
// ===== library: MasterCopy "COGNEX_OUTPUTS" =====

TYPE "COGNEX_OUTPUTS"
VERSION : 0.1
   STRUCT
      Trigger_Enable : Bool;
      Trigger : Bool;
      Reserved_0 : Bool;
      Reserved_1 : Bool;
      Reserved_2 : Bool;
      Reserved_3 : Bool;
      Reserved_4 : Bool;
      Set_Offline : Bool;
      Buffer_Results_Enable : Bool;
      Inspection_Results_Ack : Bool;
      Set_User_Data : Bool;
      Reserved_5 : Bool;
      Reserved_6 : Bool;
      Reserved_7 : Bool;
      Reserved_8 : Bool;
      Reserved_9 : Bool;
      Job_Load_ID : Byte;
      Soft_Event_0 : Bool;
      Soft_Event_1 : Bool;
      Soft_Event_2 : Bool;
      Soft_Event_3 : Bool;
      Soft_Event_4 : Bool;
      Soft_Event_5 : Bool;
      Soft_Event_6 : Bool;
      Soft_Event_7 : Bool;
      User_Data : Array[1..64] of Byte;
   END_STRUCT;
END_TYPE

// ===== library: MasterCopy "COGNEX_TO_PLC" =====

TYPE "COGNEX_TO_PLC"
VERSION : 0.1
   STRUCT
      Ready : Bool;
      NOK : Bool;
      OK : Bool;
      Program_Loaded : Byte;
      Data : Array[0..63] of Byte;
   END_STRUCT;
END_TYPE

// ===== library: MasterCopy "COGNEX_INPUTS" =====

TYPE "COGNEX_INPUTS"
VERSION : 0.1
   STRUCT
      Trigger_Ready : Bool;
      Trigger_Ack : Bool;
      Acquiring : Bool;
      Missed_Acq : Bool;
      Offline_Reason_0 : Bool;
      Offline_Reason_1 : Bool;
      Offline_Reason_2 : Bool;
      Online : Bool;
      Acquisition_ID_0 : Byte;
      Acquisition_ID_1 : Byte;
      Inspecting : Bool;
      Inspection_Completed : Bool;
      Results_Buffer_Overrun : Bool;
      Results_Valid : Bool;
      Job_Loading : Bool;
      Job_Load_Complete : Bool;
      Job_Load_Failed : Bool;
      Set_User_Data_Ack : Bool;
      Job_Pass : Bool;
      Reserved_0 : Bool;
      Reserved_1 : Bool;
      Reserved_2 : Bool;
      Reserved_3 : Bool;
      Reserved_4 : Bool;
      Reserved_5 : Bool;
      Reserved_6 : Bool;
      Current_Job_ID : Byte;
      "Inspection ID_0" : Byte;
      "Inspection ID_1" : Byte;
      "Inspection Result Code" : Word;
      "Inspection Results" : Array[0..63] of Byte;
   END_STRUCT;
END_TYPE

// ===== library: MasterCopy "PLC_TO_COGNEX" =====

TYPE "PLC_TO_COGNEX"
VERSION : 0.1
   STRUCT
      Trigger : Bool;
      Change_Program : Bool;
      Program_Number : Byte;
   END_STRUCT;
END_TYPE

// ===== library: MasterCopy "Cognex_Insight_FB" =====

// folder: 3. ST1 INSPECTION/3.2. ST1 DEVICES/3.2.0. Cognex

FUNCTION_BLOCK "Cognex_Insight_FB"   // FB52, LAD
{ S7_Optimized_Access := 'FALSE' }
VERSION : 0.1
   VAR_INPUT
      Trigger : Bool;
      Change_Program : Bool;
      Program_Number : Byte;
      Inhibit : Bool;
   END_VAR
   VAR_OUTPUT
      Ready : Bool;
      OK : Bool;
      NOK : Bool;
      Program_Loaded : Byte;
      Data : Array[0..63] of Byte;
   END_VAR
   VAR
      Inspection_Completed : Bool;
      FP_Trigger : Bool;
      FP_Inspection_completed_down : Bool;
      FP_Inspection_completed_up : Bool;
      FP_Reset_Result : Bool;
      FP_Change_Program : Bool;
      NullChar : Byte;
      Outputs : "COGNEX_OUTPUTS";
      Inputs : "COGNEX_INPUTS";
   END_VAR
   VAR_TEMP
      t_DB_NO : Int;
      In_Pointer : ANY;
      Out_Pointer : ANY;
      In_Bytes_Number : Int;
      Out_Bytes_Number : Int;
      tRetVal : Int;
   END_VAR
   VAR_TEMP   // added for the SCL form of the ladder/FBD networks
      _w1 : Bool;
      _w2 : Bool;
   END_VAR
BEGIN

REGION Network 1: TRIGGER ENABLE
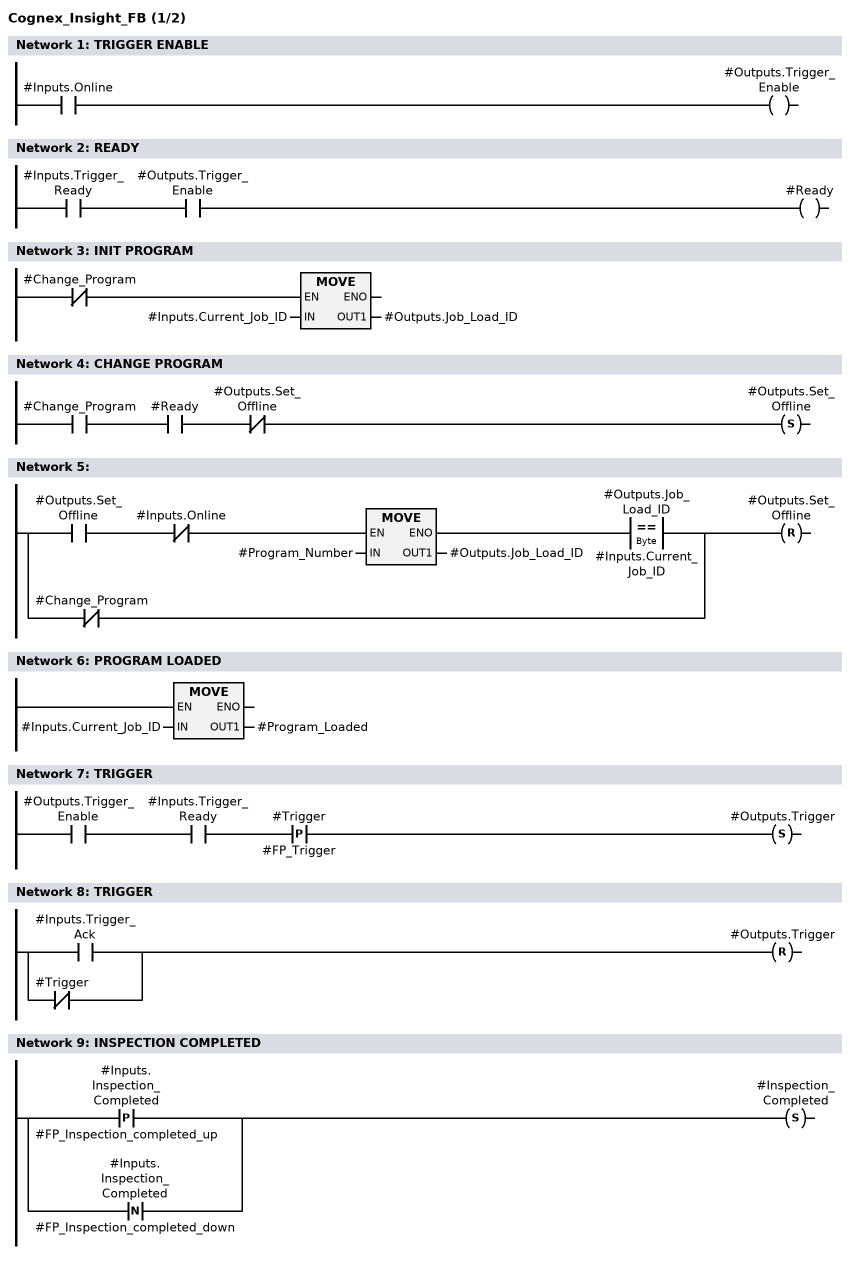
   RUNG wire#powerrail
      Contact( #Inputs.Online )
      Coil( #Outputs.Trigger_Enable )
   END_RUNG
   // the same network as SCL:
   #Outputs.Trigger_Enable := #Inputs.Online;
END_REGION

REGION Network 2: READY
   RUNG wire#powerrail
      Contact( #Inputs.Trigger_Ready )
      Contact( #Outputs.Trigger_Enable )
      Coil( #Ready )
   END_RUNG
   // the same network as SCL:
   #Ready := #Inputs.Trigger_Ready AND #Outputs.Trigger_Enable;
END_REGION

REGION Network 3: INIT PROGRAM
   RUNG wire#powerrail
      I_Contact( #Change_Program )
      { S7_GenerateENO := "TRUE" } Move(in := #Inputs.Current_Job_ID, out1 => #Outputs.Job_Load_ID)
   END_RUNG
   // the same network as SCL:
   IF NOT #Change_Program THEN #Outputs.Job_Load_ID := #Inputs.Current_Job_ID; END_IF;
END_REGION

REGION Network 4: CHANGE PROGRAM
   RUNG wire#powerrail
      Contact( #Change_Program )
      Contact( #Ready )
      I_Contact( #Outputs.Set_Offline )
      S_Coil( #Outputs.Set_Offline )
   END_RUNG
   // the same network as SCL:
   IF #Change_Program AND #Ready AND NOT #Outputs.Set_Offline THEN #Outputs.Set_Offline := TRUE; END_IF;
END_REGION

REGION Network 5
   RUNG wire#powerrail
      Contact( #Outputs.Set_Offline )
      I_Contact( #Inputs.Online )
      { S7_GenerateENO := "TRUE" } Move(in := #Program_Number, out1 => #Outputs.Job_Load_ID)
      { S7_Templates := "SrcType := Byte" } EQ_Contact(in1 := #Outputs.Job_Load_ID, in2 := #Inputs.Current_Job_ID)
      wire#w1
      R_Coil( #Outputs.Set_Offline )
   END_RUNG
   RUNG wire#powerrail
      I_Contact( #Change_Program )
   END_RUNG wire#w1
   // the same network as SCL:
   // ENO of a box is taken as its EN; it also drops when the box reports an error
   #_w1 := #Outputs.Set_Offline AND NOT #Inputs.Online;
   IF #_w1 THEN #Outputs.Job_Load_ID := #Program_Number; END_IF;
   IF (#_w1 AND (#Outputs.Job_Load_ID = #Inputs.Current_Job_ID)) OR NOT #Change_Program THEN
       #Outputs.Set_Offline := FALSE;
   END_IF;
END_REGION

REGION Network 6: PROGRAM LOADED
   RUNG wire#powerrail
      { S7_GenerateENO := "TRUE" } Move(in := #Inputs.Current_Job_ID, out1 => #Program_Loaded)
   END_RUNG
   // the same network as SCL:
   #Program_Loaded := #Inputs.Current_Job_ID;
END_REGION

REGION Network 7: TRIGGER
   RUNG wire#powerrail
      Contact( #Outputs.Trigger_Enable )
      Contact( #Inputs.Trigger_Ready )
      P_Contact(operand := #Trigger, bit := #FP_Trigger)
      S_Coil( #Outputs.Trigger )
   END_RUNG
   // the same network as SCL:
   #_w1 := #Outputs.Trigger_Enable AND #Inputs.Trigger_Ready AND #Trigger AND NOT #FP_Trigger;   // rising edge of #Trigger
   #FP_Trigger := #Trigger;
   IF #_w1 THEN #Outputs.Trigger := TRUE; END_IF;
END_REGION

REGION Network 8: TRIGGER
   RUNG wire#powerrail
      Contact( #Inputs.Trigger_Ack )
      wire#w1
      R_Coil( #Outputs.Trigger )
   END_RUNG
   RUNG wire#powerrail
      I_Contact( #Trigger )
   END_RUNG wire#w1
   // the same network as SCL:
   IF #Inputs.Trigger_Ack OR NOT #Trigger THEN #Outputs.Trigger := FALSE; END_IF;
END_REGION

REGION Network 9: INSPECTION COMPLETED
   RUNG wire#powerrail
      P_Contact(operand := #Inputs.Inspection_Completed, bit := #FP_Inspection_completed_up)
      wire#w1
      S_Coil( #Inspection_Completed )
   END_RUNG
   RUNG wire#powerrail
      N_Contact(operand := #Inputs.Inspection_Completed, bit := #FP_Inspection_completed_down)
   END_RUNG wire#w1
   // the same network as SCL:
   #_w1 := #Inputs.Inspection_Completed AND NOT #FP_Inspection_completed_up;   // rising edge of #Inputs.Inspection_Completed
   #FP_Inspection_completed_up := #Inputs.Inspection_Completed;
   #_w2 := NOT #Inputs.Inspection_Completed AND #FP_Inspection_completed_down;   // falling edge of #Inputs.Inspection_Completed
   #FP_Inspection_completed_down := #Inputs.Inspection_Completed;
   IF #_w1 OR #_w2 THEN #Inspection_Completed := TRUE; END_IF;
END_REGION

REGION Network 10: OK/NOK AND DATA / OK/NOK
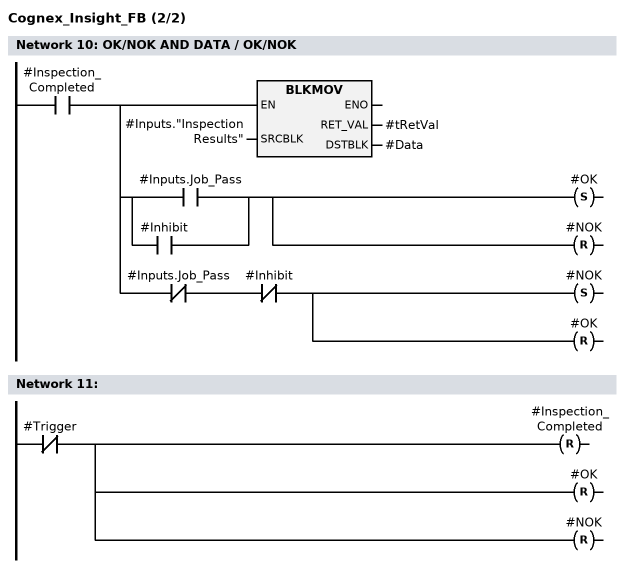
   IF #Inspection_Completed THEN
       #tRetVal := BLKMOV(SRCBLK := #Inputs."Inspection Results", DSTBLK => #Data);
   END_IF;
   IF #Inspection_Completed AND (#Inputs.Job_Pass OR #Inhibit) THEN
       #OK := TRUE;
       #NOK := FALSE;
   END_IF;
   IF #Inspection_Completed AND NOT #Inputs.Job_Pass AND NOT #Inhibit THEN
       #NOK := TRUE;
       #OK := FALSE;
   END_IF;
END_REGION

REGION Network 11
   RUNG wire#powerrail
      I_Contact( #Trigger )
      wire#w1
      R_Coil( #Inspection_Completed )
   END_RUNG
   RUNG wire#w1
      R_Coil( #OK )
   END_RUNG
   RUNG wire#w1
      R_Coil( #NOK )
   END_RUNG
   // the same network as SCL:
   IF NOT #Trigger THEN
       #Inspection_Completed := FALSE;
       #OK := FALSE;
       #NOK := FALSE;
   END_IF;
END_REGION

REGION Network 12: FUNCTION OUT
END_REGION
END_FUNCTION_BLOCK

// ===== library: MasterCopy "Keyence_SR1000_FB" =====

// folder: 3. ST1 INSPECTION/3.2. ST1 DEVICES/3.2.1. Keyence

FUNCTION_BLOCK "Keyence_SR1000_FB"   // FB59, LAD
{ S7_Optimized_Access := 'FALSE' }
VERSION : 0.1
   VAR_INPUT
      Trigger : Bool;
      Clear_Error : Bool;
      Inhibit : Bool;
   END_VAR
   VAR_OUTPUT
      Ready : Bool;
      Error : Bool;
      Error_Code : Word;
      Ok : Bool;
      NOK : Bool;
      Data : Array[0..26] of Byte;
   END_VAR
   VAR
      Inputs : "SR1000_IN";
      Outputs : "SR1000_OUT";
      "Blank Data" : Array[0..26] of Byte;
      Trigger_Flank : Bool;
      t_timeout : TON;
      s_timeout_error : Bool;
   END_VAR
   VAR_TEMP
      retval : Int;
   END_VAR
   VAR_TEMP   // added for the SCL form of the ladder/FBD networks
      _w1 : Bool;
      _w2 : Bool;
   END_VAR
BEGIN

REGION Network 1: ////////INPUTS//////////////////////
END_REGION

REGION Network 2: Ready
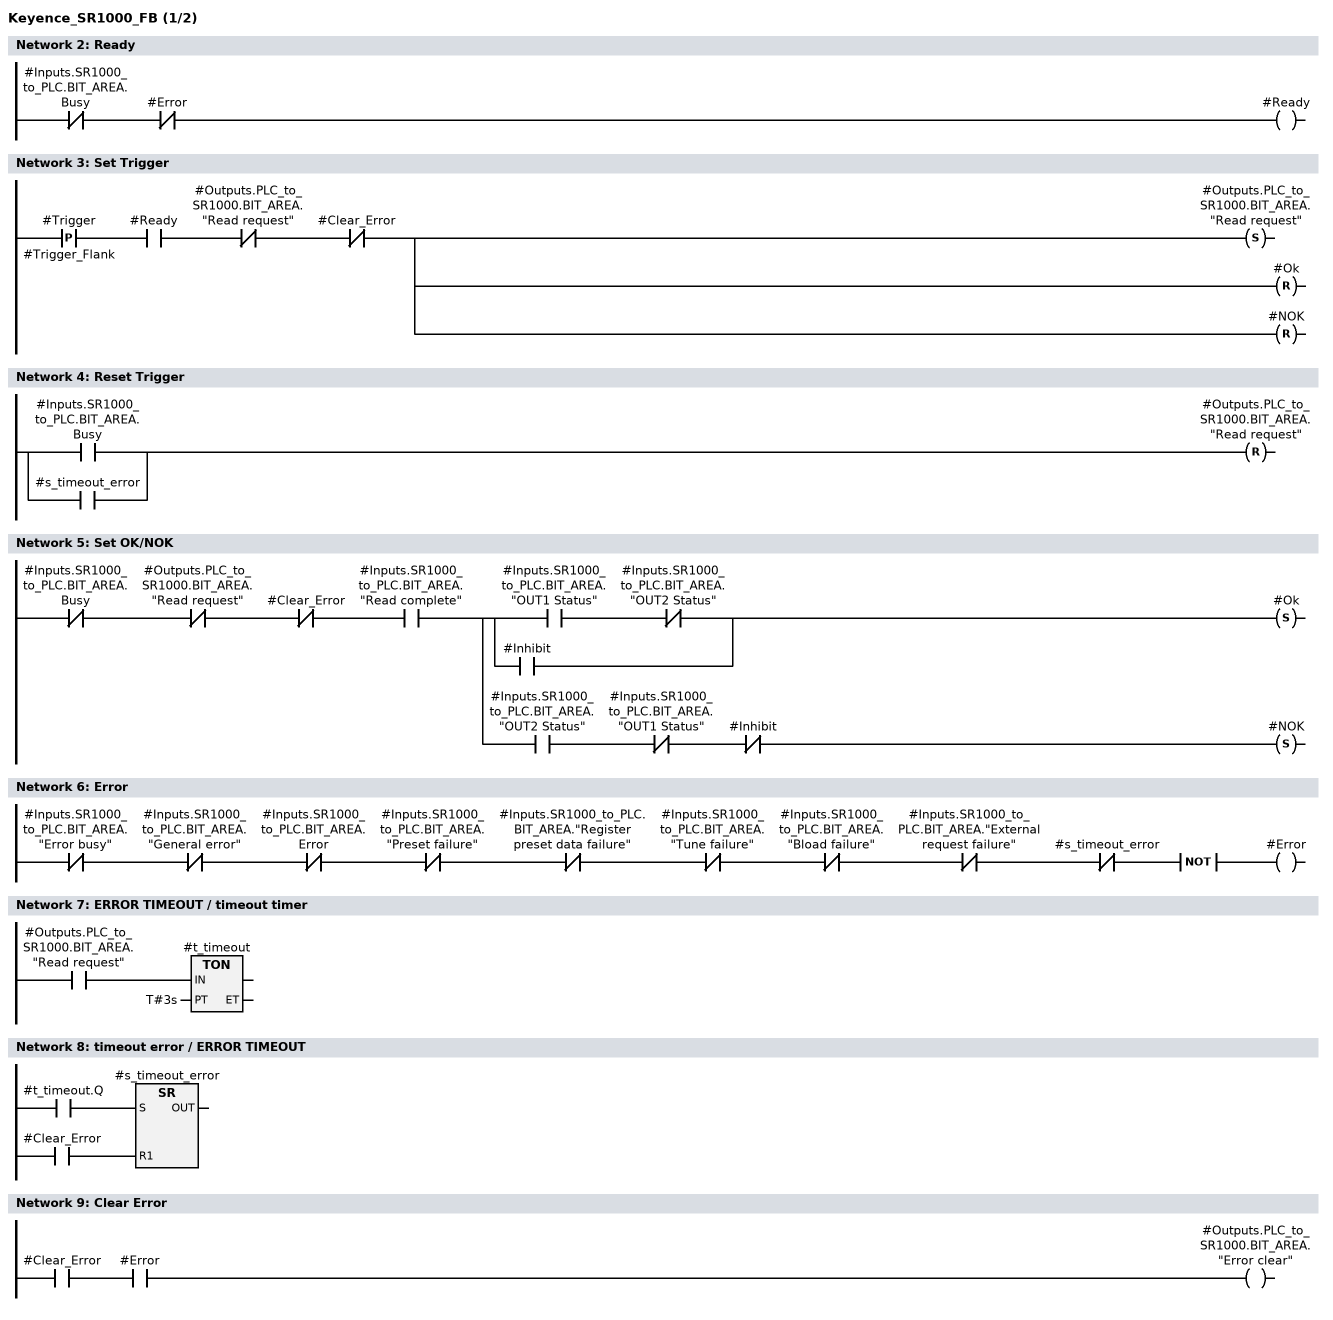
   RUNG wire#powerrail
      I_Contact( #Inputs.SR1000_to_PLC.BIT_AREA.Busy )
      I_Contact( #Error )
      Coil( #Ready )
   END_RUNG
   // the same network as SCL:
   #Ready := NOT #Inputs.SR1000_to_PLC.BIT_AREA.Busy AND NOT #Error;
END_REGION

REGION Network 3: Set Trigger
   RUNG wire#powerrail
      P_Contact(operand := #Trigger, bit := #Trigger_Flank)
      Contact( #Ready )
      I_Contact( #Outputs.PLC_to_SR1000.BIT_AREA."Read request" )
      I_Contact( #Clear_Error )
      wire#w1
      S_Coil( #Outputs.PLC_to_SR1000.BIT_AREA."Read request" )
   END_RUNG
   RUNG wire#w1
      R_Coil( #Ok )
   END_RUNG
   RUNG wire#w1
      R_Coil( #NOK )
   END_RUNG
   // the same network as SCL:
   #_w1 := #Trigger AND NOT #Trigger_Flank;   // rising edge of #Trigger
   #Trigger_Flank := #Trigger;
   #_w2 := #_w1 AND #Ready AND NOT #Outputs.PLC_to_SR1000.BIT_AREA."Read request" AND NOT #Clear_Error;
   IF #_w2 THEN
       #Outputs.PLC_to_SR1000.BIT_AREA."Read request" := TRUE;
       #Ok := FALSE;
       #NOK := FALSE;
   END_IF;
END_REGION

REGION Network 4: Reset Trigger
   RUNG wire#powerrail
      Contact( #Inputs.SR1000_to_PLC.BIT_AREA.Busy )
      wire#w1
      R_Coil( #Outputs.PLC_to_SR1000.BIT_AREA."Read request" )
   END_RUNG
   RUNG wire#powerrail
      Contact( #s_timeout_error )
   END_RUNG wire#w1
   // the same network as SCL:
   IF #Inputs.SR1000_to_PLC.BIT_AREA.Busy OR #s_timeout_error THEN
       #Outputs.PLC_to_SR1000.BIT_AREA."Read request" := FALSE;
   END_IF;
END_REGION

REGION Network 5: Set OK/NOK
   RUNG wire#powerrail
      I_Contact( #Inputs.SR1000_to_PLC.BIT_AREA.Busy )
      I_Contact( #Outputs.PLC_to_SR1000.BIT_AREA."Read request" )
      I_Contact( #Clear_Error )
      Contact( #Inputs.SR1000_to_PLC.BIT_AREA."Read complete" )
      wire#w1
      Contact( #Inputs.SR1000_to_PLC.BIT_AREA."OUT1 Status" )
      I_Contact( #Inputs.SR1000_to_PLC.BIT_AREA."OUT2 Status" )
      wire#w2
      S_Coil( #Ok )
   END_RUNG
   RUNG wire#w1
      Contact( #Inhibit )
   END_RUNG wire#w2
   RUNG wire#w1
      Contact( #Inputs.SR1000_to_PLC.BIT_AREA."OUT2 Status" )
      I_Contact( #Inputs.SR1000_to_PLC.BIT_AREA."OUT1 Status" )
      I_Contact( #Inhibit )
      S_Coil( #NOK )
   END_RUNG
   // the same network as SCL:
   #_w1 := NOT #Inputs.SR1000_to_PLC.BIT_AREA.Busy AND NOT #Outputs.PLC_to_SR1000.BIT_AREA."Read request" AND NOT #Clear_Error AND #Inputs.SR1000_to_PLC.BIT_AREA."Read complete";
   IF #_w1 AND ((#Inputs.SR1000_to_PLC.BIT_AREA."OUT1 Status" AND NOT #Inputs.SR1000_to_PLC.BIT_AREA."OUT2 Status") OR #Inhibit) THEN
       #Ok := TRUE;
   END_IF;
   IF #_w1 AND #Inputs.SR1000_to_PLC.BIT_AREA."OUT2 Status" AND NOT #Inputs.SR1000_to_PLC.BIT_AREA."OUT1 Status" AND NOT #Inhibit THEN
       #NOK := TRUE;
   END_IF;
END_REGION

REGION Network 6: Error
   RUNG wire#powerrail
      I_Contact( #Inputs.SR1000_to_PLC.BIT_AREA."Error busy" )
      I_Contact( #Inputs.SR1000_to_PLC.BIT_AREA."General error" )
      I_Contact( #Inputs.SR1000_to_PLC.BIT_AREA.Error )
      I_Contact( #Inputs.SR1000_to_PLC.BIT_AREA."Preset failure" )
      I_Contact( #Inputs.SR1000_to_PLC.BIT_AREA."Register preset data failure" )
      I_Contact( #Inputs.SR1000_to_PLC.BIT_AREA."Tune failure" )
      I_Contact( #Inputs.SR1000_to_PLC.BIT_AREA."Bload failure" )
      I_Contact( #Inputs.SR1000_to_PLC.BIT_AREA."External request failure" )
      I_Contact( #s_timeout_error )
      Not()
      Coil( #Error )
   END_RUNG
   // the same network as SCL:
   #Error := NOT (NOT #Inputs.SR1000_to_PLC.BIT_AREA."Error busy" AND NOT #Inputs.SR1000_to_PLC.BIT_AREA."General error" AND NOT #Inputs.SR1000_to_PLC.BIT_AREA.Error AND NOT #Inputs.SR1000_to_PLC.BIT_AREA."Preset failure" AND NOT #Inputs.SR1000_to_PLC.BIT_AREA."Register preset data failure" AND NOT #Inputs.SR1000_to_PLC.BIT_AREA."Tune failure" AND NOT #Inputs.SR1000_to_PLC.BIT_AREA."Bload failure" AND NOT #Inputs.SR1000_to_PLC.BIT_AREA."External request failure" AND NOT #s_timeout_error);
END_REGION

REGION Network 7: ERROR TIMEOUT / timeout timer
   #t_timeout.TON(IN := #Outputs.PLC_to_SR1000.BIT_AREA."Read request", PT := T#3s);
END_REGION

REGION Network 8: timeout error / ERROR TIMEOUT
   RUNG wire#powerrail
      Contact( #t_timeout.Q )
      S_SR(operand := #s_timeout_error, r1 := wire#w1)
   END_RUNG
   RUNG wire#powerrail
      Contact( #Clear_Error )
   END_RUNG wire#w1
   // the same network as SCL:
   IF #t_timeout.Q THEN
       #s_timeout_error := TRUE;   // SR flip-flop
   END_IF;
   IF #Clear_Error THEN #s_timeout_error := FALSE; END_IF;
END_REGION

REGION Network 9: Clear Error
   RUNG wire#powerrail
      Contact( #Clear_Error )
      Contact( #Error )
      Coil( #Outputs.PLC_to_SR1000.BIT_AREA."Error clear" )
   END_RUNG
   // the same network as SCL:
   #Outputs.PLC_to_SR1000.BIT_AREA."Error clear" := #Clear_Error AND #Error;
END_REGION

REGION Network 10: Transfer Data
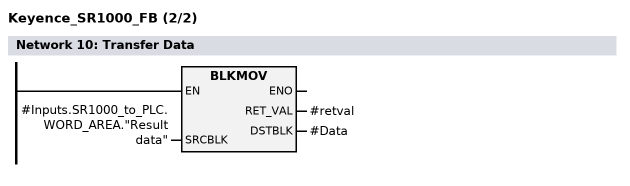
   #retval := BLKMOV(SRCBLK := #Inputs.SR1000_to_PLC.WORD_AREA."Result data", DSTBLK => #Data);
END_REGION
END_FUNCTION_BLOCK

// ===== library: MasterCopy "KEYENCE_TO_PLC" =====

TYPE "KEYENCE_TO_PLC"
   STRUCT
      Ready : Bool;
      Error : Bool;
      ErrorCode : Word;
      OK : Bool;
      NOK : Bool;
      Data : Array[0..26] of Byte;
   END_STRUCT;
END_TYPE

// ===== library: MasterCopy "PLC_TO_KEYENCE" =====

TYPE "PLC_TO_KEYENCE"
   STRUCT
      Trigger : Bool;
      "Clear Data" : Bool;
      "Clear Error" : Bool;
   END_STRUCT;
END_TYPE

// ===== library: MasterCopy "SR1000_IN" =====

TYPE "SR1000_IN"
VERSION : 0.1
   STRUCT
      SR1000_to_PLC : Struct
         BIT_AREA : Struct
            Error : Bool;   // Error
            "Result data available" : Bool;   // Result data available
            "Result data strobe" : Bool := false;   // Result data strobe
            DBX_0_3 : Bool := false;
            DBX_0_4 : Bool := false;
            DBX_0_5 : Bool := false;
            "Buffer overflow error" : Bool := false;   // Buffer overflow error
            "General error" : Bool := false;   // General error
            Busy : Bool := false;   // Busy
            "Trg busy" : Bool := false;   // Trg busy
            "Lock busy" : Bool := false;   // Lock busy
            "Mode busy" : Bool := false;   // Mode busy
            "Error busy" : Bool := false;   // Error busy
            DBX_1_5 : Bool := false;
            DBX_1_6 : Bool := false;
            DBX_1_7 : Bool := false;
            "Read complete" : Bool := false;   // Read complete
            "Preset complete" : Bool := false;   // Preset complete
            "Register preset data complete" : Bool := false;   // Register preset data complete
            "Tune complete" : Bool := false;   // Tune complete
            "Bload complete" : Bool := false;   // Bload complete
            DBX_2_5 : Bool := false;
            DBX_2_6 : Bool := false;
            "External request complete" : Bool := false;   // External request complete
            "Read failure" : Bool := false;   // Read failure
            "Preset failure" : Bool := false;   // Preset failure
            "Register preset data failure" : Bool := false;   // Register preset data failure
            "Tune failure" : Bool := false;   // Tune failure
            "Bload failure" : Bool := false;   // Bload failure
            DBX_3_5 : Bool := false;
            DBX_3_6 : Bool := false;
            "External request failure" : Bool := false;   // External request failure
            "IN1 Status" : Bool := false;   // IN1 Status
            "IN2 Status" : Bool := false;   // IN2 Status
            DBX_4_2 : Bool := false;
            DBX_4_3 : Bool := false;
            "OUT1 Status" : Bool := false;   // OUT1 Status
            "OUT2 Status" : Bool := false;   // OUT2 Status
            "OUT3 Status" : Bool := false;   // OUT3 Status
            DBX_4_7 : Bool := false;
            Unstable : Bool := false;   // Unstable
            "Matching level unstable" : Bool := false;   // Matching level unstable
            "ISO/IEC15415 unstable" : Bool := false;   // ISO/IEC15415 unstable
            "AIM DPM unstable" : Bool := false;   // AIM DPM unstable
            "SAE AS9132 unstable" : Bool := false;   // SAE AS9132 unstable
            DBX_5_5 : Bool := false;
            DBX_5_6 : Bool := false;
            DBX_5_7 : Bool := false;
         END_STRUCT;
         WORD_AREA : Struct
            "Matching level" : Word;   // Matching level
            "ISO/IEC 15415 grade" : Word;   // ISO/IEC 15415 grade
            "AIM DPM Grade" : Word;   // AIM DPM Grade
            DBW_7_3 : Word;
            "Read result code" : Word;   // Read result code
            "Preset result code" : Word;   // Preset result code
            "Register preset data result code" : Word;   // Register preset data result code
            "Tune result code" : Word;   // Tune result code
            "Bload result code" : Word;   // Bload result code
            DBW_8_5 : Word;
            DBW_8_6 : Word;
            "Ext. request result code" : Word;   // Ext. request result code
            "General error code" : Word;   // General error code
            "Slave ID" : Word;   // Slave ID
            "Result data ready count" : Word;   // Result data ready count
            "Result data update count" : Word;   // Result data update count
            "Trigger input count for master" : Word;   // Trigger input count for master
            DBW_9_4 : Byte;   // Result data size
            "Result data size" : Byte;
            "Result data" : Array[1..128] of Byte;   // Result data
         END_STRUCT;
      END_STRUCT;
   END_STRUCT;
END_TYPE

// ===== library: MasterCopy "SR1000_OUT" =====

TYPE "SR1000_OUT"
VERSION : 0.1
   STRUCT
      PLC_to_SR1000 : Struct
         BIT_AREA : Struct
            DBX170_0 : Bool;
            "Result data latch" : Bool := false;   // Result data latch
            DBX170_2 : Bool := false;
            DBX170_3 : Bool := false;
            DBX170_4 : Bool := false;
            DBX170_5 : Bool := false;
            DBX170_6 : Bool := false;
            "Error clear" : Bool := false;   // Error clear
            "Read request" : Bool := false;   // Read request
            "Preset request" : Bool := false;   // Preset request
            "Register preset" : Bool := false;   // Register preset
            "Tune request" : Bool := false;   // Tune request
            "Bload request" : Bool := false;   // Bload request
            DBX171_5 : Bool := false;
            DBX171_6 : Bool := false;
            DBX171_7 : Bool := false;
            "Read complete clear" : Bool := false;   // Read complete clear
            "Preset complet clear" : Bool := false;   // Preset complet clear
            "Register preset data complete clear" : Bool := false;   // Register preset data complete clear
            "Tune complete clear" : Bool := false;   // Tune complete clear
            "Bload complete clear" : Bool := false;   // Bload complete clear
            DBX172_5 : Bool := false;
            DBX172_6 : Bool := false;
            "External request complete clear" : Bool := false;   // External request complete clear
            "Bank number\Bload file number" : Word;   // Bank number\Bload file number
            "User data size" : Word := 16#0;   // User data size
            "User data" : Array[1..128] of Byte;   // User data
         END_STRUCT;
      END_STRUCT;
   END_STRUCT;
END_TYPE

// ===== library: MasterCopy "DATAMAN_TO_PLC" =====

TYPE "DATAMAN_TO_PLC"
VERSION : 0.1
   STRUCT
      Ready : Bool;
      Trigger_ACK : Bool;
      OK : Bool;
      NOK : Bool;
      Error : Bool;
      Result_ID : Word;
      Result_Lenght : Int;
      Result : Array[1..64] of Byte;
   END_STRUCT;
END_TYPE

// ===== library: MasterCopy "DATAMAN_INPUTS" =====

TYPE "DATAMAN_INPUTS"
VERSION : 0.1
   STRUCT
      Trigger_Ready : Bool;
      Trigger_Ack : Bool;
      Acquiring : Bool;
      Missed_Acq : Bool;
      Reserved_0 : Bool;
      Reserved_1 : Bool;
      Reserved_2 : Bool;
      Reserved_3 : Bool;
      Trigger_ID_0 : Byte;
      Trigger_ID_1 : Byte;
      Decoding : Bool;
      Decode_Complete : Bool;
      Result_Buffer_Overrun : Bool;
      Result_Available : Bool;
      Reserved_4 : Bool;
      Reserved_5 : Bool;
      Reserved_6 : Bool;
      General_Fault : Bool;
      Train_Code_Ack : Bool;
      Train_Match_String_Ack : Bool;
      Train_Focus_Ack : Bool;
      Train_Brightness_Ack : Bool;
      Ultrain_Ack : Bool;
      Reserved_7 : Bool;
      Execute_DMCC_Ack : Bool;
      Set_Match_String_Ack : Bool;
      Result_ID_0 : Byte;
      Result_ID_1 : Byte;
      Result_Code_0 : Byte;
      Result_Code_1 : Byte;
      Result_Extended_0 : Byte;
      Result_Extended_1 : Byte;
      Result_Length_0 : Byte;
      Result_Length_1 : Byte;
      Result_Data_0 : Byte;
      Result_Data_1 : Byte;
      Result_Data_2 : Byte;
      Result_Data_3 : Byte;
      Result_Data_4 : Byte;
      Result_Data_5 : Byte;
      Result_Data_6 : Byte;
      Result_Data_7 : Byte;
      Result_Data_8 : Byte;
      Result_Data_9 : Byte;
      Result_Data_10 : Byte;
      Result_Data_11 : Byte;
      Result_Data_12 : Byte;
      Result_Data_13 : Byte;
      Result_Data_14 : Byte;
      Result_Data_15 : Byte;
      Result_Data_16 : Byte;
      Result_Data_17 : Byte;
      Result_Data_18 : Byte;
      Result_Data_19 : Byte;
      Result_Data_20 : Byte;
      Result_Data_21 : Byte;
      Result_Data_22 : Byte;
      Result_Data_23 : Byte;
      Result_Data_24 : Byte;
      Result_Data_25 : Byte;
      Result_Data_26 : Byte;
      Result_Data_27 : Byte;
      Result_Data_28 : Byte;
      Result_Data_29 : Byte;
      Result_Data_30 : Byte;
      Result_Data_31 : Byte;
      Result_Data_32 : Byte;
      Result_Data_33 : Byte;
      Result_Data_34 : Byte;
      Result_Data_35 : Byte;
      Result_Data_36 : Byte;
      Result_Data_37 : Byte;
      Result_Data_38 : Byte;
      Result_Data_39 : Byte;
      Result_Data_40 : Byte;
      Result_Data_41 : Byte;
      Result_Data_42 : Byte;
      Result_Data_43 : Byte;
      Result_Data_44 : Byte;
      Result_Data_45 : Byte;
      Result_Data_46 : Byte;
      Result_Data_47 : Byte;
      Result_Data_48 : Byte;
      Result_Data_49 : Byte;
      Result_Data_50 : Byte;
      Result_Data_51 : Byte;
      Result_Data_52 : Byte;
      Result_Data_53 : Byte;
      Result_Data_54 : Byte;
      Result_Data_55 : Byte;
      Result_Data_56 : Byte;
      Result_Data_57 : Byte;
      Result_Data_58 : Byte;
      Result_Data_59 : Byte;
      Result_Data_60 : Byte;
      Result_Data_61 : Byte;
      Result_Data_62 : Byte;
      Result_Data_63 : Byte;
   END_STRUCT;
END_TYPE

// ===== library: MasterCopy "DATAMAN_OUTPUTS" =====

TYPE "DATAMAN_OUTPUTS"
VERSION : 0.1
   STRUCT
      Trigger_Enable : Bool;
      Trigger : Bool;
      Reserved_0 : Bool;
      Reserved_1 : Bool;
      Reserved_2 : Bool;
      Reserved_3 : Bool;
      Reserved_4 : Bool;
      Reserved_5 : Bool;
      Result_Buffer_Enable : Bool;
      Results_Ack : Bool;
      Reserved_6 : Bool;
      Reserved_7 : Bool;
      Reserved_8 : Bool;
      Reserved_9 : Bool;
      Reserved_10 : Bool;
      Reserved_11 : Bool;
      Train_Code : Bool;
      Train_Match_String : Bool;
      Train_Focus : Bool;
      Train_Brightness : Bool;
      Ultrain : Bool;
      Reserved_12 : Bool;
      Execute_DMCC : Bool;
      Set_Match_String : Bool;
      User_Data_Option_0 : Byte;
      User_Data_Option_1 : Byte;
      User_Data_Lenght_0 : Byte;
      User_Data_Lenght_1 : Byte;
      User_Data_0 : Byte;
      User_Data_1 : Byte;
      User_Data_2 : Byte;
      User_Data_3 : Byte;
      User_Data_4 : Byte;
      User_Data_5 : Byte;
      User_Data_6 : Byte;
      User_Data_7 : Byte;
      User_Data_8 : Byte;
      User_Data_9 : Byte;
      User_Data_10 : Byte;
      User_Data_11 : Byte;
      User_Data_12 : Byte;
      User_Data_13 : Byte;
      User_Data_14 : Byte;
      User_Data_15 : Byte;
      User_Data_16 : Byte;
      User_Data_17 : Byte;
      User_Data_18 : Byte;
      User_Data_19 : Byte;
      User_Data_20 : Byte;
      User_Data_21 : Byte;
      User_Data_22 : Byte;
      User_Data_23 : Byte;
      User_Data_24 : Byte;
      User_Data_25 : Byte;
      User_Data_26 : Byte;
      User_Data_27 : Byte;
      User_Data_28 : Byte;
      User_Data_29 : Byte;
      User_Data_30 : Byte;
      User_Data_31 : Byte;
      User_Data_32 : Byte;
      User_Data_33 : Byte;
      User_Data_34 : Byte;
      User_Data_35 : Byte;
      User_Data_36 : Byte;
      User_Data_37 : Byte;
      User_Data_38 : Byte;
      User_Data_39 : Byte;
      User_Data_40 : Byte;
      User_Data_41 : Byte;
      User_Data_42 : Byte;
      User_Data_43 : Byte;
      User_Data_44 : Byte;
      User_Data_45 : Byte;
      User_Data_46 : Byte;
      User_Data_47 : Byte;
      User_Data_48 : Byte;
      User_Data_49 : Byte;
      User_Data_50 : Byte;
      User_Data_51 : Byte;
      User_Data_52 : Byte;
      User_Data_53 : Byte;
      User_Data_54 : Byte;
      User_Data_55 : Byte;
      User_Data_56 : Byte;
      User_Data_57 : Byte;
      User_Data_58 : Byte;
      User_Data_59 : Byte;
      User_Data_60 : Byte;
      User_Data_61 : Byte;
      User_Data_62 : Byte;
      User_Data_63 : Byte;
   END_STRUCT;
END_TYPE

// ===== library: MasterCopy "PLC_TO_DATAMAN" =====

TYPE "PLC_TO_DATAMAN"
VERSION : 0.1
   STRUCT
      Reset : Bool;
      Result_Ack : Bool;
   END_STRUCT;
END_TYPE

// ===== library: MasterCopy "Dataman_FB" =====

// folder: 8. DRAWERS/8.2. ST6 DEVICES/8.2.1.Dataman

FUNCTION_BLOCK "Dataman_FB"   // FB51, LAD
{ S7_Optimized_Access := 'FALSE' }
VERSION : 0.1
   VAR_INPUT
      Reset : Bool;
      I_O_Address : Int;   // dirección entradas salidas en configuración de hardware
      DB_NO : Int;   // Número del db de instancia
   END_VAR
   VAR_OUTPUT
      Ready : Bool;
      Trigger_ACK : Bool;
      OK : Bool;
      NOK : Bool;
      Error : Bool;
      Result_ID : Word;
      Result_Lenght : Int;
      Result : Array[1..64] of Byte;
   END_VAR
   VAR
      WaitingNewTrigger : Bool;
      ResultAckPending : Bool;
      Result_Code : Word;
      Inputs : "DATAMAN_INPUTS";
      Outputs : "DATAMAN_OUTPUTS";
   END_VAR
   VAR_TEMP
      On : Bool;
      Off : Bool;
      t_DB_NO : Int;
      In_Pointer : ANY;
      Outputs_Bytes_Number : Int;
      Inputs_Bytes_Number : Int;
      Out_Pointer : ANY;
      tRetVal : Int;
   END_VAR
   VAR_TEMP   // added for the SCL form of the ladder/FBD networks
      _w1 : Bool;
   END_VAR
BEGIN

REGION Network 1
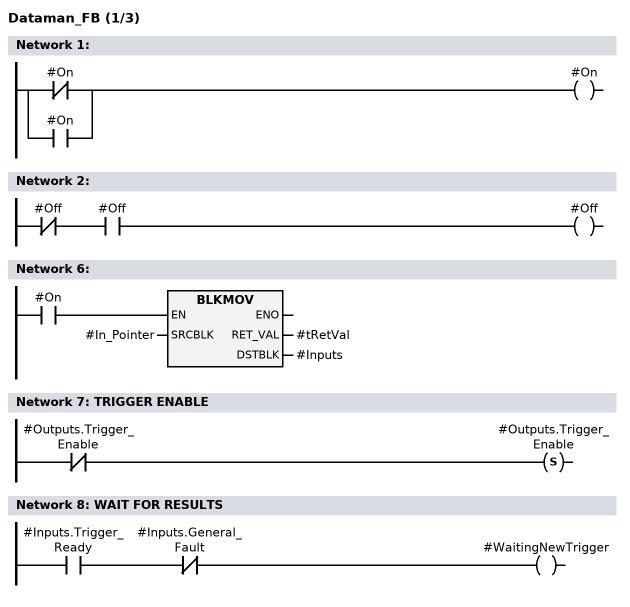
   RUNG wire#powerrail
      I_Contact( #On )
      wire#w1
      Coil( #On )
   END_RUNG
   RUNG wire#powerrail
      Contact( #On )
   END_RUNG wire#w1
   // the same network as SCL:
   #On := NOT #On OR #On;
END_REGION

REGION Network 2
   RUNG wire#powerrail
      I_Contact( #Off )
      Contact( #Off )
      Coil( #Off )
   END_RUNG
   // the same network as SCL:
   #Off := NOT #Off AND #Off;
END_REGION

REGION Network 3 (STL)

         L     #DB_NO;
         T     #t_DB_NO;
         OPN   DB[ #t_DB_NO];
END_REGION

REGION Network 4 (STL)

         L     77;
         T     #Inputs_Bytes_Number;
END_REGION

REGION Network 5 (STL)
   //En primer lugar, apuntar al puntero
         LAR1;
   //Carga de parámetros en los bytes del puntero
   //Byte 0 = 10h para S7
         L     16#10;
         T     LB[AR1, P#0.0];

   //Byte 1 = Tipo de datos
   //02h para byte
         L     16#02;
         T     LB[AR1, P#1.0];

   //Byte2-Byte3 (int) = Factor de repetición
   //número de bytes (tipo de datos) a mover
         L     #Inputs_Bytes_Number;
         T     LW[AR1, P#2.0];

   //Byt42-Byte5 (int) = Número de DB
   //0 en este caso porque no se trata de DB
         L     0;
         T     LW[AR1, P#4.0];

   //En los siguientes 4 bytes van el area de memoria y la dirección inicial
   //Se borra inicialmente
         L     0;
         T     LD[AR1, P#6.0];

   //Byte 6 = Area de memoria
   //81h para entradas
         L     16#81;
         T     LB[AR1, P#6.0];


   //Byte7-Byte9 (int) = dirección (byte.bit)
   //ver formato
         L     #I_O_Address;
         SLW   3;
         T     LW[AR1, P#8.0];
END_REGION

REGION Network 6
   IF #On THEN #tRetVal := BLKMOV(SRCBLK := #In_Pointer, DSTBLK => #Inputs); END_IF;
END_REGION

REGION Network 7: TRIGGER ENABLE
   RUNG wire#powerrail
      I_Contact( #Outputs.Trigger_Enable )
      S_Coil( #Outputs.Trigger_Enable )
   END_RUNG
   // the same network as SCL:
   IF NOT #Outputs.Trigger_Enable THEN #Outputs.Trigger_Enable := TRUE; END_IF;
END_REGION

REGION Network 8: WAIT FOR RESULTS
   RUNG wire#powerrail
      Contact( #Inputs.Trigger_Ready )
      I_Contact( #Inputs.General_Fault )
      Coil( #WaitingNewTrigger )
   END_RUNG
   // the same network as SCL:
   #WaitingNewTrigger := #Inputs.Trigger_Ready AND NOT #Inputs.General_Fault;
END_REGION

REGION Network 9: SAVE DATA
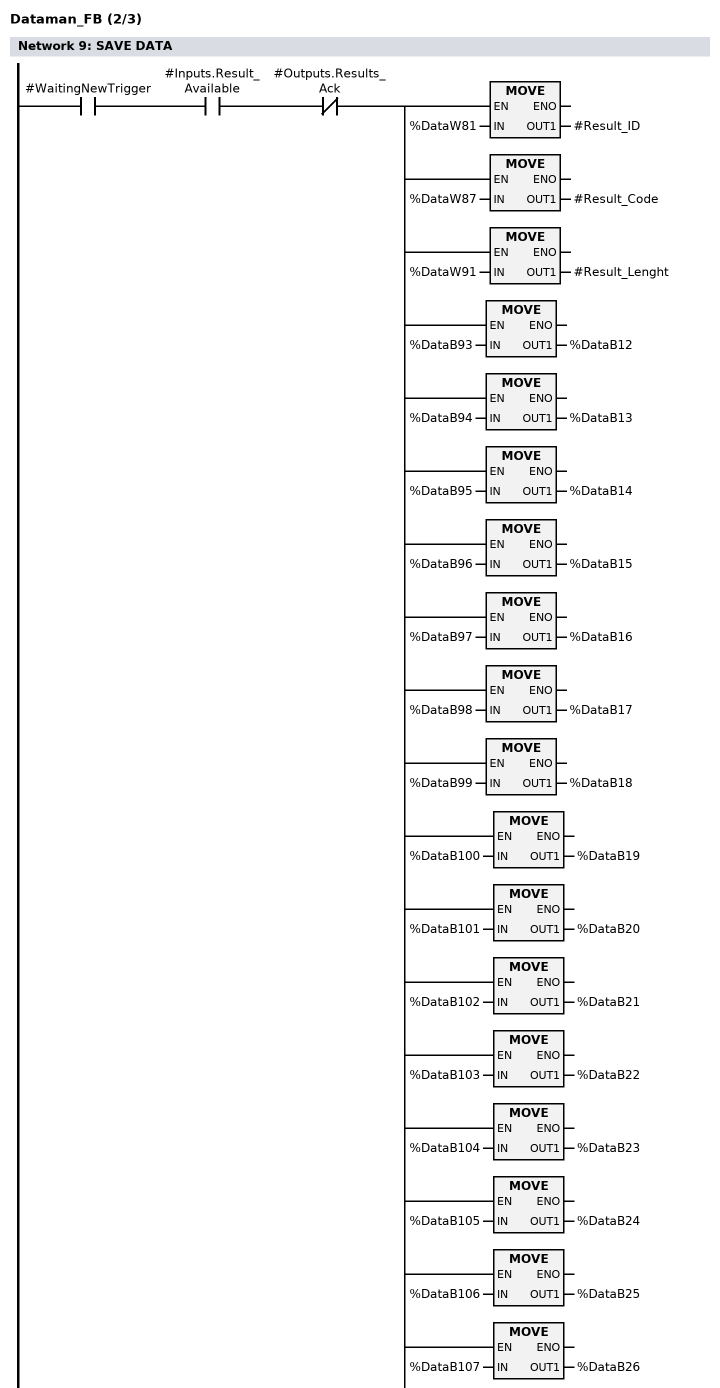
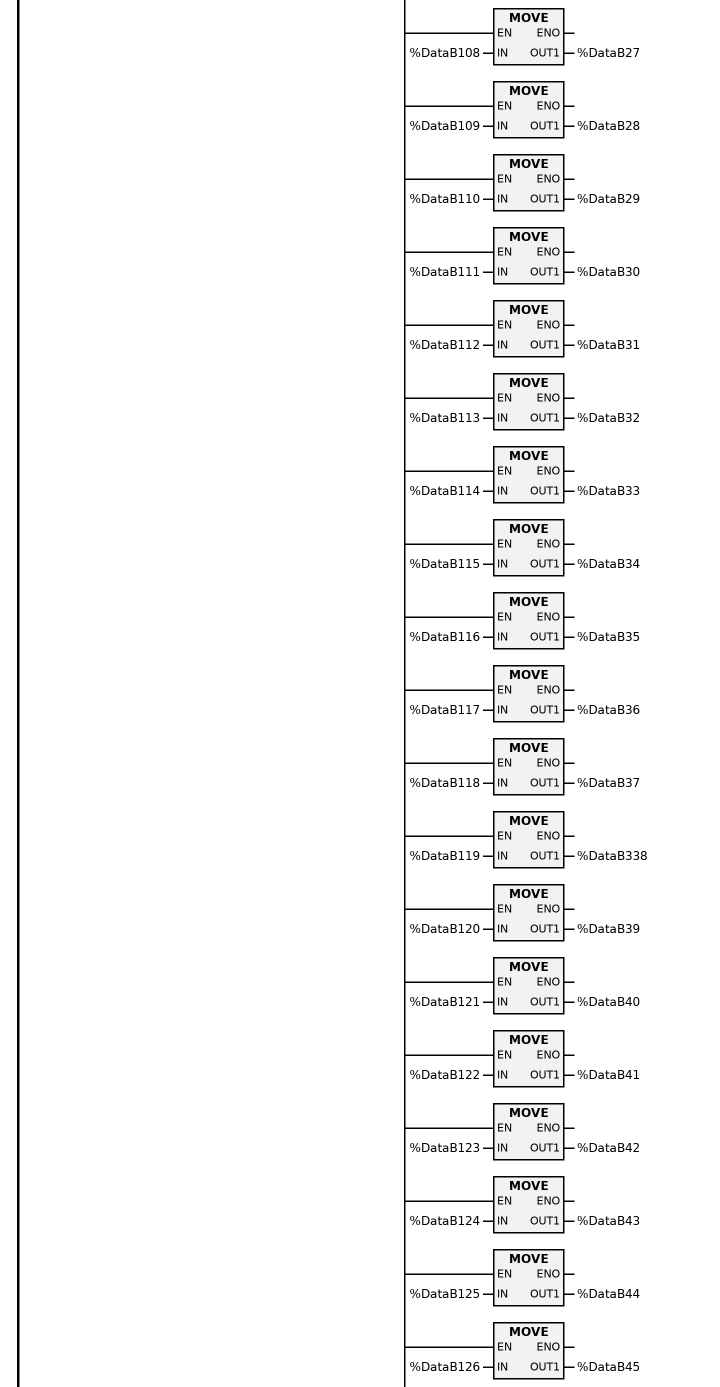
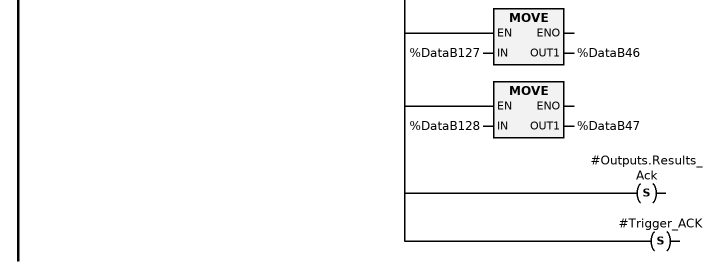
   RUNG wire#powerrail
      Contact( #WaitingNewTrigger )
      Contact( #Inputs.Result_Available )
      I_Contact( #Outputs.Results_Ack )
      wire#w1
      { S7_GenerateENO := "TRUE" } Move(in := %DataW81, out1 => #Result_ID)
   END_RUNG
   RUNG wire#w1
      { S7_GenerateENO := "TRUE" } Move(in := %DataW87, out1 => #Result_Code)
   END_RUNG
   RUNG wire#w1
      { S7_GenerateENO := "TRUE" } Move(in := %DataW91, out1 => #Result_Lenght)
   END_RUNG
   RUNG wire#w1
      { S7_GenerateENO := "TRUE" } Move(in := %DataB93, out1 => %DataB12)
   END_RUNG
   RUNG wire#w1
      { S7_GenerateENO := "TRUE" } Move(in := %DataB94, out1 => %DataB13)
   END_RUNG
   RUNG wire#w1
      { S7_GenerateENO := "TRUE" } Move(in := %DataB95, out1 => %DataB14)
   END_RUNG
   RUNG wire#w1
      { S7_GenerateENO := "TRUE" } Move(in := %DataB96, out1 => %DataB15)
   END_RUNG
   RUNG wire#w1
      { S7_GenerateENO := "TRUE" } Move(in := %DataB97, out1 => %DataB16)
   END_RUNG
   RUNG wire#w1
      { S7_GenerateENO := "TRUE" } Move(in := %DataB98, out1 => %DataB17)
   END_RUNG
   RUNG wire#w1
      { S7_GenerateENO := "TRUE" } Move(in := %DataB99, out1 => %DataB18)
   END_RUNG
   RUNG wire#w1
      { S7_GenerateENO := "TRUE" } Move(in := %DataB100, out1 => %DataB19)
   END_RUNG
   RUNG wire#w1
      { S7_GenerateENO := "TRUE" } Move(in := %DataB101, out1 => %DataB20)
   END_RUNG
   RUNG wire#w1
      { S7_GenerateENO := "TRUE" } Move(in := %DataB102, out1 => %DataB21)
   END_RUNG
   RUNG wire#w1
      { S7_GenerateENO := "TRUE" } Move(in := %DataB103, out1 => %DataB22)
   END_RUNG
   RUNG wire#w1
      { S7_GenerateENO := "TRUE" } Move(in := %DataB104, out1 => %DataB23)
   END_RUNG
   RUNG wire#w1
      { S7_GenerateENO := "TRUE" } Move(in := %DataB105, out1 => %DataB24)
   END_RUNG
   RUNG wire#w1
      { S7_GenerateENO := "TRUE" } Move(in := %DataB106, out1 => %DataB25)
   END_RUNG
   RUNG wire#w1
      { S7_GenerateENO := "TRUE" } Move(in := %DataB107, out1 => %DataB26)
   END_RUNG
   RUNG wire#w1
      { S7_GenerateENO := "TRUE" } Move(in := %DataB108, out1 => %DataB27)
   END_RUNG
   RUNG wire#w1
      { S7_GenerateENO := "TRUE" } Move(in := %DataB109, out1 => %DataB28)
   END_RUNG
   RUNG wire#w1
      { S7_GenerateENO := "TRUE" } Move(in := %DataB110, out1 => %DataB29)
   END_RUNG
   RUNG wire#w1
      { S7_GenerateENO := "TRUE" } Move(in := %DataB111, out1 => %DataB30)
   END_RUNG
   RUNG wire#w1
      { S7_GenerateENO := "TRUE" } Move(in := %DataB112, out1 => %DataB31)
   END_RUNG
   RUNG wire#w1
      { S7_GenerateENO := "TRUE" } Move(in := %DataB113, out1 => %DataB32)
   END_RUNG
   RUNG wire#w1
      { S7_GenerateENO := "TRUE" } Move(in := %DataB114, out1 => %DataB33)
   END_RUNG
   RUNG wire#w1
      { S7_GenerateENO := "TRUE" } Move(in := %DataB115, out1 => %DataB34)
   END_RUNG
   RUNG wire#w1
      { S7_GenerateENO := "TRUE" } Move(in := %DataB116, out1 => %DataB35)
   END_RUNG
   RUNG wire#w1
      { S7_GenerateENO := "TRUE" } Move(in := %DataB117, out1 => %DataB36)
   END_RUNG
   RUNG wire#w1
      { S7_GenerateENO := "TRUE" } Move(in := %DataB118, out1 => %DataB37)
   END_RUNG
   RUNG wire#w1
      { S7_GenerateENO := "TRUE" } Move(in := %DataB119, out1 => %DataB338)
   END_RUNG
   RUNG wire#w1
      { S7_GenerateENO := "TRUE" } Move(in := %DataB120, out1 => %DataB39)
   END_RUNG
   RUNG wire#w1
      { S7_GenerateENO := "TRUE" } Move(in := %DataB121, out1 => %DataB40)
   END_RUNG
   RUNG wire#w1
      { S7_GenerateENO := "TRUE" } Move(in := %DataB122, out1 => %DataB41)
   END_RUNG
   RUNG wire#w1
      { S7_GenerateENO := "TRUE" } Move(in := %DataB123, out1 => %DataB42)
   END_RUNG
   RUNG wire#w1
      { S7_GenerateENO := "TRUE" } Move(in := %DataB124, out1 => %DataB43)
   END_RUNG
   RUNG wire#w1
      { S7_GenerateENO := "TRUE" } Move(in := %DataB125, out1 => %DataB44)
   END_RUNG
   RUNG wire#w1
      { S7_GenerateENO := "TRUE" } Move(in := %DataB126, out1 => %DataB45)
   END_RUNG
   RUNG wire#w1
      { S7_GenerateENO := "TRUE" } Move(in := %DataB127, out1 => %DataB46)
   END_RUNG
   RUNG wire#w1
      { S7_GenerateENO := "TRUE" } Move(in := %DataB128, out1 => %DataB47)
   END_RUNG
   RUNG wire#w1
      S_Coil( #Outputs.Results_Ack )
   END_RUNG
   RUNG wire#w1
      S_Coil( #Trigger_ACK )
   END_RUNG
   // the same network as SCL:
   IF #WaitingNewTrigger AND #Inputs.Result_Available AND NOT #Outputs.Results_Ack THEN
       #Result_ID := %DataW81;
       #Result_Code := %DataW87;
       #Result_Lenght := %DataW91;
       %DataB12 := %DataB93;
       %DataB13 := %DataB94;
       %DataB14 := %DataB95;
       %DataB15 := %DataB96;
       %DataB16 := %DataB97;
       %DataB17 := %DataB98;
       %DataB18 := %DataB99;
       %DataB19 := %DataB100;
       %DataB20 := %DataB101;
       %DataB21 := %DataB102;
       %DataB22 := %DataB103;
       %DataB23 := %DataB104;
       %DataB24 := %DataB105;
       %DataB25 := %DataB106;
       %DataB26 := %DataB107;
       %DataB27 := %DataB108;
       %DataB28 := %DataB109;
       %DataB29 := %DataB110;
       %DataB30 := %DataB111;
       %DataB31 := %DataB112;
       %DataB32 := %DataB113;
       %DataB33 := %DataB114;
       %DataB34 := %DataB115;
       %DataB35 := %DataB116;
       %DataB36 := %DataB117;
       %DataB37 := %DataB118;
       %DataB338 := %DataB119;
       %DataB39 := %DataB120;
       %DataB40 := %DataB121;
       %DataB41 := %DataB122;
       %DataB42 := %DataB123;
       %DataB43 := %DataB124;
       %DataB44 := %DataB125;
       %DataB45 := %DataB126;
       %DataB46 := %DataB127;
       %DataB47 := %DataB128;
   END_IF;
   #_w1 := #WaitingNewTrigger AND #Inputs.Result_Available AND NOT #Outputs.Results_Ack;
   IF #_w1 THEN
       #Outputs.Results_Ack := TRUE;
       #Trigger_ACK := TRUE;
   END_IF;
END_REGION

REGION Network 10: RESET RESULTS ACKNOWLEDGE SIGNAL AS SOON AS I IS RECOGNIZED BY READER
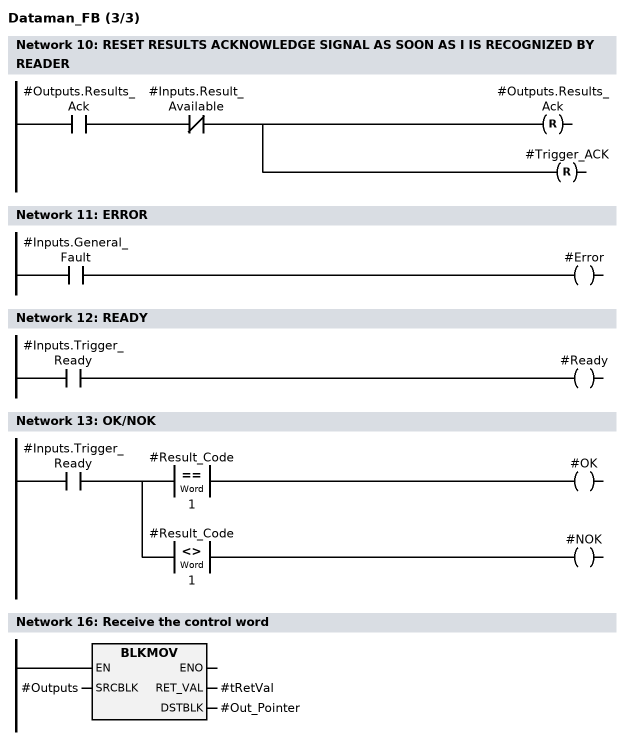
   RUNG wire#powerrail
      Contact( #Outputs.Results_Ack )
      I_Contact( #Inputs.Result_Available )
      wire#w1
      R_Coil( #Outputs.Results_Ack )
   END_RUNG
   RUNG wire#w1
      R_Coil( #Trigger_ACK )
   END_RUNG
   // the same network as SCL:
   #_w1 := #Outputs.Results_Ack AND NOT #Inputs.Result_Available;
   IF #_w1 THEN
       #Outputs.Results_Ack := FALSE;
       #Trigger_ACK := FALSE;
   END_IF;
END_REGION

REGION Network 11: ERROR
   RUNG wire#powerrail
      Contact( #Inputs.General_Fault )
      Coil( #Error )
   END_RUNG
   // the same network as SCL:
   #Error := #Inputs.General_Fault;
END_REGION

REGION Network 12: READY
   RUNG wire#powerrail
      Contact( #Inputs.Trigger_Ready )
      Coil( #Ready )
   END_RUNG
   // the same network as SCL:
   #Ready := #Inputs.Trigger_Ready;
END_REGION

REGION Network 13: OK/NOK
   RUNG wire#powerrail
      Contact( #Inputs.Trigger_Ready )
      wire#w1
      { S7_Templates := "SrcType := Word" } EQ_Contact(in1 := #Result_Code, in2 := 1)
      Coil( #OK )
   END_RUNG
   RUNG wire#w1
      { S7_Templates := "SrcType := Word" } NE_Contact(in1 := #Result_Code, in2 := 1)
      Coil( #NOK )
   END_RUNG
   // the same network as SCL:
   #OK := #Inputs.Trigger_Ready AND (#Result_Code = 1);
   #NOK := #Inputs.Trigger_Ready AND (#Result_Code <> 1);
END_REGION

REGION Network 14 (STL)

         L     71;
         T     #Outputs_Bytes_Number;
END_REGION

REGION Network 15 (STL)
   //En primer lugar, apuntar al puntero
         LAR1;
   //Carga de parámetros en los bytes del puntero
   //Byte 0 = 10h para S7
         L     16#10;
         T     LB[AR1, P#0.0];

   //Byte 1 = Tipo de datos
   //02h para byte
         L     16#02;
         T     LB[AR1, P#1.0];

   //Byte2-Byte3 (int) = Factor de repetición
   //número de bytes (tipo de datos) a mover
         L     #Outputs_Bytes_Number;
         T     LW[AR1, P#2.0];

   //Byt42-Byte5 (int) = Número de DB
   //0 en este caso porque no se trata de DB
         L     0;
         T     LW[AR1, P#4.0];

   //En los siguientes 4 bytes van el area de memoria y la dirección inicial
   //Se borra inicialmente
         L     0;
         T     LD[AR1, P#6.0];

   //Byte 6 = Area de memoria
   //82h para salidas
         L     16#82;
         T     LB[AR1, P#6.0];


   //Byte7-Byte9 (int) = dirección (byte.bit)
   //ver formato
         L     #I_O_Address;
         SLW   3;
         T     LW[AR1, P#8.0];
END_REGION

REGION Network 16: Receive the control word
   #tRetVal := BLKMOV(SRCBLK := #Outputs, DSTBLK => #Out_Pointer);
END_REGION
END_FUNCTION_BLOCK

// ===== library: MasterCopy "SINA_POS" =====

// folder: AxisControl

FUNCTION_BLOCK "SINA_POS"   // FB600, SCL
TITLE = 'Positioning with SINAMICS and S7'
{ S7_Optimized_Access := 'TRUE' }
AUTHOR : DRVDPS7
FAMILY : DRIVES
NAME : SINA_POS
VERSION : 5.7
// Copyright (C) Siemens AG 2012. All Rights Reserved. Confidential
// -------------------------------------------------------------------------------------- 
// SINA_POS: Positionierung mit dem Antriebsbaustein SINAMICS S120/G120 <-> S7-1200
// ------------------------------------------------------------------------------------- Ersteller: Siemens AG Erlangen A&D MC PM   Datum:  07.07.10        Vers.:2.1
// Änderung:  J.B. Typical Team                       18.12.12              2.2
//     Umsetzung in SCL / TIA 
// Änderung:  J.B. Typical Team                       18.04.13              2.3
//     Bei Betriebsart "Referenzieren - Referenzpunkt setzen"
//     nicht intern setzen sondern Eingang #Execute abfragen als 
//     Startbedingung
// Änderung:  J.B. Typical Team                       29.04.13              2.4
//     1. Off1 möglich bei ungültige Betriebsart
//     2. Referenzpunkt setzen Exceute übernehmen
//     3. Fehlermeldung ausgeben bei Wechel ohne 
//        Beendigung der Betriebsart 
//     4. "Q" an den Ausgänge entfernen
//     5. Neuer Ausgang PwrInhibit
//      
// Änderung:  J.B. Typical Team                       14.05.13              2.5
//     Fehlerbehebung und Defaultwerte ändern
// Änderung:  J.B. Typical Team                       28.06.13              2.6
//     HW-Zugriffsermittlung über LOG2MOD
// Änderung:  J.B. Typical Team                       18.07.13              2.7
//     HW-Zugriffsermittlung über zwei HW-Eingänge
// Änderung:  J.B. Typical Team                       18.09.13              2.8
//     Konvertierungsfehler behoben
// Änderung:  J.B. Typical Team                       25.09.13              2.9
//     Bei Betriebswechsel von 3 nach 6 darf MidStart nicht sitzen
// Änderung:  J.B. Typical Team                       31.03.14              3.0
//     In der Betriebsart 1-3 und 6 darf MidTrTyp nicht sitzen
// Änderung:  J.B. Typical Team                       25.06.14              3.1
//     Das Quittierbit "AckFlt" immer durchreichen
// Änderung:  J.B. Typical Team                       30.07.14              4.0
//     Festlegung auf einheitlicher neuer Version 4.0
// Änderung:  J.B. Typical Team                       07.11.14              4.1
//     Fehlerbehebung falsche Zuweisung von Off1 bei Mode 4
//     und Mode 8(DriveLib V4 - RQ 346046)
// Änderung:  F.G. Typical Team                       16.04.15              4.2
//     Anzahl der Zyklen die auf die Rückmeldung fliegendes Ref.
//     gewartet wird verdoppelt (siRetryMax = 10)  (DriveLib V4 - RQ 367986)
// Änderung:  F.G. Typical Team                       15.09.15              4.3
//     Anzahl der Zyklen die auf die Rückmeldung fliegendes Ref.
//     gewartet noch einmal um 5 erhöht (siRetryMax = 15)  (DriveLib V4 - RQ 367986)
// Änderung:  F.G. Typical Team                       15.09.15              4.4
//     Abfrage des richtigen Bits im EPosZSW1 (Zeile 1394)es muss das Bit12 
//     und nicht das Bit 11 abgefragt werden  (DriveLib V4 - RQ 367986)
// Änderung:  F.G. Typical Team                       03.12.15              4.5
//     1. Ein-/Ausgänge an Programmierleitfaden für TIA-Portal angepasst
//        Zusätzlicher Eingang um alle Bits in den STWs zu bedienen
//     2. Warnung durch Initialisierung elimininiert
// Änderung:  F.G. Typical Team                       13.09.16              4.6
//     Ausgabewerte am Ausgang "Status" angepasst 
// 
// Änderung:  G.F. Typical Team                       11.01.17              5.0
//     - Festlegung auf einheitlicher neuer Version 5.0 
// 
// Änderung:  G.F. Typical Team                       13.07.17              5.1
//     - Zuordnung der Bits von ConfigPos korrigiert 
// 
// Änderung:  G.F. Typical Team                       12.01.18              5.2
//     - RQ2637983 sxSendBuf.EPosSTW2.%X1 in Mode 7 und 8 rücksetzen 
// Änderung:  G.F. Typical Team                       20.07.18              5.3
//     - ZSW1.13 als Ausgang zur Verfügung gestellt (wegen FW - Änderung)
// Änderung:  G.F. Typical Team                       18.10.18              5.4
//     - RQ 824321 Zähler für fliegendes Referenzieren zurücksetzen
// Änderung:  G.F. Typical Team                       08.02.19              5.5
//     - Version wegen Änderungen in älteren Lib-Versionen 
// Änderung:  G.F. Typical Team                       08.02.19              5.6
//     - RQ 3901129 Fehler Flankenauswertung Eingang ExecuteMode behoben Bibliothek V7
// Änderung:  G.F. Typical Team                       17.05.19              5.7
//     - RQ 4094299 Fehler Referenzfahrt wird nicht gestartet behoben Bibliothek V7
// Funktion: Positionierung mit dem Antriebsbaustein SINAMICS S120/G120 <-> S7-1200
// ********************************************************************************************************************************************************
// ************************************************************************FB283***************************************************************************
// ********************************************************************************************************************************************************
// Copyright (C) Siemens AG 2012. All Rights Reserved. Confidential
// -------------------------------------------------------------------------------------- 
// SINA_POS: Positionierung mit dem Antriebsbaustein SINAMICS S120/G120 <-> S7-1200
// ------------------------------------------------------------------------------------- Ersteller: Siemens AG Erlangen A&D MC PM   Datum:  07.07.10        Vers.:2.1
// Änderung:  J.B. Typical Team                       18.12.12              2.2
//     Umsetzung in SCL / TIA 
// Änderung:  J.B. Typical Team                       18.04.13              2.3
//     Bei Betriebsart "Referenzieren - Referenzpunkt setzen"
//     nicht intern setzen sondern Eingang #Execute abfragen als 
//     Startbedingung
// Änderung:  J.B. Typical Team                       29.04.13              2.4
//     1. Off1 möglich bei ungültige Betriebsart
//     2. Referenzpunkt setzen Exceute übernehmen
//     3. Fehlermeldung ausgeben bei Wechel ohne 
//        Beendigung der Betriebsart 
//     4. "Q" an den Ausgänge entfernen
//     5. Neuer Ausgang PwrInhibit
//      
// Änderung:  J.B. Typical Team                       14.05.13              2.5
//     Fehlerbehebung und Defaultwerte ändern
// Änderung:  J.B. Typical Team                       28.06.13              2.6
//     HW-Zugriffsermittlung über LOG2MOD
// Änderung:  J.B. Typical Team                       18.07.13              2.7
//     HW-Zugriffsermittlung über zwei HW-Eingänge
// Änderung:  J.B. Typical Team                       18.09.13              2.8
//     Konvertierungsfehler behoben
// Änderung:  J.B. Typical Team                       25.09.13              2.9
//     Bei Betriebswechsel von 3 nach 6 darf MidStart nicht sitzen
// Änderung:  J.B. Typical Team                       31.03.14              3.0
//     In der Betriebsart 1-3 und 6 darf MidTrTyp nicht sitzen
// Änderung:  J.B. Typical Team                       25.06.14              3.1
//     Das Quittierbit "AckFlt" immer durchreichen
// Änderung:  J.B. Typical Team                       30.07.14              4.0
//     Festlegung auf einheitlicher neuer Version 4.0
// Änderung:  J.B. Typical Team                       07.11.14              4.1
//     Fehlerbehebung falsche Zuweisung von Off1 bei Mode 4
//     und Mode 8(DriveLib V4 - RQ 346046)
// Änderung:  F.G. Typical Team                       16.04.15              4.2
//     Anzahl der Zyklen die auf die Rückmeldung fliegendes Ref.
//     gewartet wird verdoppelt (siRetryMax = 10)  (DriveLib V4 - RQ 367986)
// Änderung:  F.G. Typical Team                       15.09.15              4.3
//     Anzahl der Zyklen die auf die Rückmeldung fliegendes Ref.
//     gewartet noch einmal um 5 erhöht (siRetryMax = 15)  (DriveLib V4 - RQ 367986)
// Änderung:  F.G. Typical Team                       15.09.15              4.4
//     Abfrage des richtigen Bits im EPosZSW1 (Zeile 1394)es muss das Bit12 
//     und nicht das Bit 11 abgefragt werden  (DriveLib V4 - RQ 367986)
// Änderung:  F.G. Typical Team                       03.12.15              4.5
//     1. Ein-/Ausgänge an Programmierleitfaden für TIA-Portal angepasst
//        Zusätzlicher Eingang um alle Bits in den STWs zu bedienen
//     2. Warnung durch Initialisierung elimininiert
// Änderung:  F.G. Typical Team                       13.09.16              4.6
//     Ausgabewerte am Ausgang "Status" angepasst 
// 
// Änderung:  G.F. Typical Team                       11.01.17              5.0
//     - Festlegung auf einheitlicher neuer Version 5.0 
// 
// Änderung:  G.F. Typical Team                       13.07.17              5.1
//     - Zuordnung der Bits von ConfigPos korrigiert 
// 
// Änderung:  G.F. Typical Team                       12.01.18              5.2
//     - RQ2637983 sxSendBuf.EPosSTW2.%X1 in Mode 7 und 8 rücksetzen 
// Änderung:  G.F. Typical Team                       20.07.18              5.3
//     - ZSW1.13 als Ausgang zur Verfügung gestellt (wegen FW - Änderung)
// Änderung:  G.F. Typical Team                       18.10.18              5.4
//     - RQ 824321 Zähler für fliegendes Referenzieren zurücksetzen
// Änderung:  G.F. Typical Team                       08.02.19              5.5
//     - Version wegen Änderungen in älteren Lib-Versionen 
// Änderung:  G.F. Typical Team                       08.02.19              5.6
//     - RQ 3901129 Fehler Flankenauswertung Eingang ExecuteMode behoben Bibliothek V7
// Funktion: Positionierung mit dem Antriebsbaustein SINAMICS S120/G120 <-> S7-1200
// ********************************************************************************************************************************************************
// ************************************************************************FB283***************************************************************************
// ********************************************************************************************************************************************************
   VAR_INPUT
      ModePos : Int := 0;   // Settings of the mode / Auswahl EPos Betriebsart (0= keine; 1,2,3 = MDI; 4,5 = Referenzieren; 6= Verfarhsätze; 7,8 = Tippen)
      EnableAxis : Bool := 0;   // 1 = Enable the drive / 0-->1 = Einschalten des Antriebs (OFF1 = 0-->1)
      CancelTraversing : Bool := 1;   // 0 = Reject active traverse task / 0 = Abruch der laufenden Verfahrbewegung (1=kein Abbruch)
      IntermediateStop : Bool := 1;   // 0 = Intermediate STOP of traverse command / 0 = Zwischenhalt der laufenden Verfahrbewegung (1= kein Zwischenhalt)
      Positive : Bool := 0;   // 1 = Direction positive / 1 = Positive Verfahrrichtung
      Negative : Bool := 0;   // 1 = Direction negative / 1 = Negative Verfahrrichtung
      Jog1 : Bool := 0;   // 1 = Use jog 1 (direction / speed) / 1 = Tippen Sollwert 1 auswählen
      Jog2 : Bool := 0;   // 1 = Use jog 2 (direction / speed) / 1 = Tippen Sollwert 2 auswählen
      FlyRef : Bool := 0;   // 1 = Start flying reference function / 1 = Aktivierung Fliegendes Referenzieren (nicht möglich bei ModePos = 4, 5)
      AckError : Bool := 0;   // 1 = Acknowledge of errors / 1 = Achs / EPos Fehlerquittierung anwählen
      ExecuteMode : Bool := 0;   // 0-->1 = Start the mode / 0-->1 = Starten der mit ModePos gewählten Betriebsart
      Position : Real := 0.0;   // Position of the MDI mode or setting of traversing block / Positionssollwert [LU] für Direkt Sollwert vorgabe (MDI)
      Velocity : DInt := 0;   // MDI velocity / MDI Geschwindigkeit [1000*LU / min]
      OverV : Int := 100;   // Override of velocity in [%] --> 4000h=100% / Geschwindigkeit Skalierung (Alle Betriebsarten 4000h = 100%))
      OverAcc : Int := 100;   // Override of acceleration in [%] --> 4000h=100% / MDI Beschleunigung (4000h = 100%)
      OverDec : Int := 100;   // Override of deceleration in [%] --> 4000h=100% / MDI Verzögerung (4000h = 100%)
      ConfigEPos : DWord := 16#0000_0003;   // binary programmed input to control all functions in the telegram without its own function block input / Binärcodierter Eingang zur Ansteuerung aller nicht als Bausteineingang verfügbaren Steuerbits
      HWIDSTW : HW_IO := 0;   // Hardware Identifer set point slot / Hardware Identifer des Sollwert Slots
      HWIDZSW : HW_IO := 0;   // Hardware Identifer actual value slot / Hardware Identifer des Istwert Slots
      RefTorque : Real;
      RefSpeed : Real;
      Factor : Real;   // Virgulden sonraki basamak
      SoftPosTlr : Real;   // Softpos OK Toleransı
   END_VAR
   VAR_OUTPUT
      AxisEnabled : Bool := 0;   // 1= Axis in operation / 1= EPos Achse ist in Betrieb
      AxisPosOk : Bool := 0;   // 1= Position setpoint reached / 1= EPos Achsposition erreicht
      SoftPosOK : Bool;
      AxisSpFixed : Bool := 0;   // 1= Setpoint fixed (Attention: Dependence on SINAMICS firmware) / 1= Sollwert steht (Achtung: Abhängigkeit von SINAMICS Firmware)
      AxisRef : Bool := 0;   // 1= Reference point set / 1= EPos Achse referenziert
      AxisWarn : Bool := 0;   // 1= Axis alarm / warning present / 1= Antriebswarnung aktiv
      AxisError : Bool := 0;   // 1= Axis fault present / 1= Antriebs / EPos Fehler vorhanden
      Lockout : Bool := 0;   // 1= Axis in lockout state / 1= Einschaltsperre aktiv
      ActVelocity : Real := 0.0;   // Actual drive speed (has to be normed with p2000 --> 40000000h = 100%) / Aktuelle Geschwindigkeit (40000000h = 100% von p2000 in [rpm])
      ActPosition : Real := 0.0;   // Actual position in [LU] / Aktuelle Position in LU
      ActMode : Int := 0;   // Active EPos mode / Aktuellle Betriebsart
      EPosZSW1 : Word := 0;   // Status of EPOS ZSW1
      EPosZSW2 : Word := 0;   // Status of EPOS ZSW2
      ActWarn : Word := 0;   // Actual number of warning / Aktuelle Warnung
      ActFault : Word := 0;   // Actual number of error / Aktuelle Störung
      Error : Bool := 0;   // 1 = Error (FB and Infeed) / Fehler (Antrieb und / oder Funktionsbaustein)
      Status : Word := 0;   // Status output (7002 = FB in operation; 8xxx = error description - read the manual) / Statusausgabe (7002 = FB in Betrieb; 8xxx = Feherbeschreibung siehe Doku)
      DiagID : Word := 0;   // Error codes of the cyclic system funtion blocks DPWR / DPRD_DAT / Fehlercode der zyklischen Systemfunktionen DPWR / DPRD_DAT
      Torque : Real;
   END_VAR
   VAR
      sbOff1Edge : Bool := 0;   // Positive edge of starting or stopping the device
      sbOff1 : Bool := 0;   // Starting or stopping the device
      sbExecuteEdge : Bool := 0;   // Positive edge of activate traversing block
      sbExecute : Bool := 0;   // Activate traversing block
      sbRefTypEdge : Bool := 0;   // Positive edge of referencing type "flying reference"
      sbRefTyp : Bool := 0;   // Referencing type "flying reference"
      sbMdiStart : Bool := 0;   // Direct setpoint input / MDI - start
      sbMdiStartEdge : Bool := 0;   // Positive edge of direct setpoint input / MDI - start
      sbRefStart : Bool := 0;   // Referencing start
      sbJogInc : Bool := 0;   // Jogging incremental
      sbReady : Bool := 0;   // Ready to power up / to start
      sbIOp : Bool := 0;   // Ready to operate
      sbAccel : Bool := 0;   // Axis accelerating
      sbDecel : Bool := 0;   // Axis decelerating
      sbAlarm : Bool := 0;   // Alarm / Warnung present
      sbFault : Bool := 0;   // Fault present
      sbFWD : Bool := 0;   // Axis drives forwards
      sbBWD : Bool := 0;   // Axis drives backwards
      sbBusy : Bool := 0;   // Mode of operation is explained
      swStatus : Word := 16#0000;   // Mode of operation disturbance
      swEPosZSW1 : Word := 16#0000;   // Status of EPOS ZSW1 / EPos Zustandswort 1
      swEPosZSW2 : Word := 16#0000;   // Status of EPOS ZSW2 / EPos Zustandswort 2
      siExecuteCyc : Int := 0;   // Counter of runcycle of active traversing block
      siRefTypCyc : Int := 0;   // Counter of runcycle of referencing type "flying reference"
      siJogIncCyc : Int := 0;   // Counter of runcycle of jogging incremental
      siMdiStartCyc : Int := 0;   // Counter of runcycle of direct setpoint input / MDI - start
      siRefActRetry : Int := 0;   // Counter of retry of reference point approach active
      siModePos : Int := 0;   // Setting of mode
      siModePosMax : Int := 8;   // Max. count of mode
      siCycWait : Int := 5;   // Counter of cycle of waiting
      siRetryMax : Int := 30;   // Max. count of cycles of retry
      sbModePos : Bool := 0;   // Mode of setting okay
      sxSendBuf : Struct   // send buffer of telegram for sending data to the drive
         STW1 : Word := WORD#16#0000;   // STW1sxSTW1 : STRUCT Jog1 : BOOL:=0; // ST-Wort-1 Bit 08 --> 1 = Jogging - signal source 1 Jog2 : BOOL:=0; // ST-Wort-1 Bit 09 --> 1 = Jogging - signal source 2 LB : BOOL:=1; // Allways // ST-Wort-1 Bit 10 --> 1 = Life bit RefStart : BOOL:=0; // ST-Wort-1 Bit 11 --> 1 = Referencing start / stop Bit12 : BOOL:=0; // ST-Wort-1 Bit 12 --> 1 = Reserve Bit13 : BOOL:=0; // ST-Wort-1 Bit 13 --> 1 = Externer Satzwechsel Bit14 : BOOL:=0; // ST-Wort-1 Bit 14 --> 1 = Reserve Bit15 : BOOL:=0; // ST-Wort-1 Bit 15 --> 1 = Reserve Off1 : BOOL:=0; // ST-Wort-1 Bit 00 --> 1 = OFF1/ON (flanks acceptance) Off2 : BOOL:=1; // Allways // ST-Wort-1 Bit 01 --> 1 = OFF2/ON (enable possible) Off3 : BOOL:=1; // Allways // ST-Wort-1 Bit 02 --> 1 = OFF3/ON (enable possible) Enc : BOOL:=1; // Allways // ST-Wort-1 Bit 03 --> 1 = Enable controller RejTrvTsk : BOOL:=0; // ST-Wort-1 Bit 04 --> 1 = Traversing block and MDI - reject task IntMStop : BOOL:=0; // ST-Wort-1 Bit 05 --> 1 = Traversing block and MDI - intermediate - STOP TrvStart : BOOL:=0; // ST-Wort-1 Bit 06 --> 1 = Traversing start - direct setpoint input / MDI - transfer edge AckFault : BOOL:=0; // ST-Wort-1 Bit 07 --> 1 = Acknowledge fault END_STRUCT;
         EPosSTW1 : Word := WORD#16#0000;   // EPOSSTW1sxEPosSTW1 : STRUCT MdiTyp : BOOL:=0; // EPOS-Wort-1 Bit 08 --> 1 = Direct setpoint input / MDI - positioning type MdiPos : BOOL:=0; // EPOS-Wort-1 BIT 09 --> 1 = Direct setpoint input / MDI - positive direction MdiNeg : BOOL:=0; // EPOS-Wort-1 BIT 10 --> 1 = Direct setpoint input / MDI - negative direction Bit11 : BOOL:=0; // EPOS-Wort-1 BIT 11 --> 1 = Reserve MdiTrTyp : BOOL:=0; // EPOS-Wort-1 BIT 12 --> 1 = Direct setpoint input / MDI - transfer type Bit13 : BOOL:=0; // EPOS-Wort-1 BIT 13 --> 1 = Reserve MdiSetup : BOOL:=0; // EPOS-Wort-1 BIT 14 --> 1 = Direct setpoint input / MDI - setup selection MdiStart : BOOL:=0; // EPOS-Wort-1 BIT 15 --> 1 = Direct setpoint input / MDI - start TrvBit0 : BOOL:=0; // EPOS-Wort-1 BIT 00 --> 1 = Traversing block - block selection bit 0 TrvBit1 : BOOL:=0; // EPOS-Wort-1 BIT 01 --> 1 = Traversing block - block selection bit 1 TrvBit2 : BOOL:=0; // EPOS-Wort-1 BIT 02 --> 1 = Traversing block - block selection bit 2 TrvBit3 : BOOL:=0; // EPOS-Wort-1 BIT 03 --> 1 = Traversing block - block selection bit 3 TrvBit4 : BOOL:=0; // EPOS-Wort-1 BIT 04 --> 1 = Traversing block - block selection bit 4 TrvBit5 : BOOL:=0; // EPOS-Wort-1 Bit 05 --> 1 = Traversing block - block selection bit 5 Bit06 : BOOL:=0; // EPOS-Wort-1 Bit 06 --> 1 = Reserve Bit07 : BOOL:=0; // EPOS-Wort-1 Bit 07 --> 1 = Reserve END_STRUCT;
         EPosSTW2 : Word := WORD#16#0000;   // EPOSSTW2sxEPosSTW2 : STRUCT RefTyp : BOOL:=0; // EPOS-Wort-2 Bit 08 --> 1 = Referencing type RefStDi : BOOL:=0; // EPOS-Wort-2 Bit 09 --> 1 = Homing start direction RefInpS : BOOL:=0; // EPOS-Wort-2 Bit 10 --> 1 = Referencing passive - input selection RefEdge : BOOL:=0; // EPOS-Wort-2 Bit 11 --> 1 = Referencing passive - edge evaluation Bit12 : BOOL:=0; // EPOS-Wort-2 Bit 12 --> 1 = Reserve Bit13 : BOOL:=0; // EPOS-Wort-2 Bit 13 --> 1 = Reserve SftLimAct : BOOL:=0; // EPOS-Wort-2 Bit 14 --> 1 = Software limit switch activation StpCamAct : BOOL:=0; // EPOS-Wort-2 Bit 15 --> 1 = Stop output cam activation TrkMode : BOOL:=0; // EPOS-Wort-2 Bit 00 --> 1 = Tracking mode active SetRefPt : BOOL:=0; // EPOS-Wort-2 Bit 01 --> 1 = Set reference point ActRefCam : BOOL:=0; // EPOS-Wort-2 Bit 02 --> 1 = Reference cam active Bit03 : BOOL:=0; // EPOS-Wort-2 Bit 03 --> 1 = Reserve Bit04 : BOOL:=0; // EPOS-Wort-2 Bit 04 --> 1 = Reserve JogInc : BOOL:=0; // EPOS-Wort-2 Bit 05 --> 1 = Jogging - jogging incremental Bit06 : BOOL:=0; // EPOS-Wort-2 Bit 06 --> 1 = Reserve Bit07 : BOOL:=0; // EPOS-Wort-2 Bit 07 --> 1 = Reserve END_STRUCT;
         STW2 : Word := WORD#16#0000;   // STW2sxSTW2 : STRUCT TrvFixStp : BOOL:=0; // ST-Wort-2 Bit 08 --> 1 = Travel fixed STOP GlbTrgCom : BOOL:=0; // ST-Wort-2 Bit 09 --> 1 = Global trigger command Bit10 : BOOL:=0; // ST-Wort-2 Bit 10 --> 1 = Reserve MotSwOver : BOOL:=0; // ST-Wort-2 Bit 11 --> 1 = Motor switch over finished MsZykBit0 : BOOL:=0; // ST-Wort-2 Bit 12 --> 1 = Master life bit 0 MsZykBit1 : BOOL:=0; // ST-Wort-2 Bit 13 --> 1 = Master life bit 1 MsZykBit2 : BOOL:=0; // ST-Wort-2 Bit 14 --> 1 = Master life bit 2 MsZykBit3 : BOOL:=0; // ST-Wort-2 Bit 15 --> 1 = Master life bit 3 DDSBit0 : BOOL:=0; // ST-Wort-2 Bit 00 --> 1 = Drive data set bit 0 DDSBit1 : BOOL:=0; // ST-Wort-2 Bit 01 --> 1 = Drive data set bit 1 DDSBit2 : BOOL:=0; // ST-Wort-2 Bit 02 --> 1 = Drive data set bit 2 DDSBit3 : BOOL:=0; // ST-Wort-2 Bit 03 --> 1 = Drive data set bit 3 DDSBit4 : BOOL:=0; // ST-Wort-2 Bit 04 --> 1 = Drive data set bit 4 GlbStart : BOOL:=0; // ST-Wort-2 Bit 05 --> 1 = Global start ResIComp : BOOL:=0; // ST-Wort-2 Bit 06 --> 1 = Reset I-component of speed controller ActPrkAxis : BOOL:=0; // ST-Wort-2 Bit 07 --> 1 = Activate parking axis END_STRUCT;
         OverrideV : Word := WORD#16#0000;   // Velocity override
         Position : DWord := DWORD#16#0000_0000;   // Setpoint of position
         Velocity : DWord := DWORD#16#0000_0000;   // Setpoint of velocity
         OverrideA : Word := WORD#16#0000;   // Accelerating override
         OverrideD : Word := WORD#16#0000;   // Decelerating override
         Reserve : Word := WORD#16#0000;   // Reserve
      END_STRUCT;
      sxRecvBuf : Struct   // receive buffer of telegram for receiving data from the drive
         ZSW1 : Word := WORD#16#0000;   // ZSW1sxZSW1 : STRUCT NoFlwErr : BOOL:=0; // ZSW-Wort-1 Bit 08 --> 1 = Following error in tolerance LbCr : BOOL:=0; // ZSW-Wort-1 Bit 09 --> 1 = Lifebit control request TargPos : BOOL:=0; // ZSW-Wort-1 Bit 10 --> 1 = Target position reached RefPSet : BOOL:=0; // ZSW-Wort-1 Bit 11 --> 1 = Reference point set TrvTskAck : BOOL:=0; // ZSW-Wort-1 Bit 12 --> 1 = Traversing task acknowledge StndStill : BOOL:=0; // ZSW-Wort-1 Bit 13 --> 1 = [n_ist] < Drehzahlsollwert 3 Accel : BOOL:=0; // ZSW-Wort-1 Bit 14 --> 1 = Axis accelerating Decel : BOOL:=0; // ZSW-Wort-1 Bit 15 --> 1 = Axis decelerating RTS : BOOL:=0; // ZSW-Wort-1 Bit 00 --> 1 = Ready to power up / to start RDY : BOOL:=0; // ZSW-Wort-1 Bit 01 --> 1 = Ready to operate IOp : BOOL:=0; // ZSW-Wort-1 Bit 02 --> 1 = In operation (operation enabled) Fault : BOOL:=0; // ZSW-Wort-1 Bit 03 --> 1 = Fault present NoOff2Act : BOOL:=0; // ZSW-Wort-1 Bit 04 --> 1 = OFF2 inactive NoOff3Act : BOOL:=0; // ZSW-Wort-1 Bit 05 --> 1 = OFF3 inactive PowInhbt : BOOL:=0; // ZSW-Wort-1 Bit 06 --> 1 = Power ON inhibit active Alarm : BOOL:=0; // ZSW-Wort-1 Bit 07 --> 1 = Alarm / Warning present END_STRUCT;
         EPosZSW1 : Word := WORD#16#0000;   // EPOSZSW1sxEPosZSW1 : STRUCT StpCamMinAct : BOOL:=0; // EPOS-Wort-1 Bit 08 --> 1 = STOP cam minus active StpCamPlsAct : BOOL:=0; // EPOS-Wort-1 Bit 09 --> 1 = STOP cam plus active JogAct : BOOL:=0; // EPOS-Wort-1 Bit 10 --> 1 = Jogging active RefAct : BOOL:=0; // EPOS-Wort-1 Bit 11 --> 1 = Reference point approach active FlyRefAct : BOOL:=0; // EPOS-Wort-1 Bit 12 --> 1 = Flying referencing active TrvBlAct : BOOL:=0; // EPOS-Wort-1 Bit 13 --> 1 = Traversing block active MdiStupAct : BOOL:=0; // EPOS-Wort-1 Bit 14 --> 1 = MDI setup active MdiPosAct : BOOL:=0; // EPOS-Wort-1 Bit 15 --> 1 = MDI positing active ActTrvBit0 : BOOL:=0; // EPOS-Wort-1 BIT 00 --> 1 = Active traversing block bit 0 ActTrvBit1 : BOOL:=0; // EPOS-Wort-1 Bit 01 --> 1 = Active traversing block bit 1 ActTrvBit2 : BOOL:=0; // EPOS-Wort-1 Bit 02 --> 1 = Active traversing block bit 2 ActTrvBit3 : BOOL:=0; // EPOS-Wort-1 Bit 03 --> 1 = Active traversing block bit 3 ActTrvBit4 : BOOL:=0; // EPOS-Wort-1 Bit 04 --> 1 = Active traversing block bit 4 ActTrvBit5 : BOOL:=0; // EPOS-Wort-1 Bit 05 --> 1 = Active traversing block bit 5 Bit06 : BOOL:=0; // EPOS-Wort-1 Bit 06 --> 1 = Reserve Bit07 : BOOL:=0; // EPOS-Wort-1 Bit 07 --> 1 = Reserve END_STRUCT;
         EPosZSW2 : Word := WORD#16#0000;   // EPOSZSW2sxEPosZSW2 : STRUCT PosSmCam1 : BOOL:=0; // EPOS-Wort-2 Bit 08 --> 1 = Position actual value <= cam position 1 PosSmCam2 : BOOL:=0; // EPOS-Wort-2 Bit 09 --> 1 = Position actual value <= cam position 2 TrvOut1 : BOOL:=0; // EPOS-Wort-2 Bit 10 --> 1 = Direct output 1 via traversing block TrvOut2 : BOOL:=0; // EPOS-Wort-2 Bit 11 --> 1 = Direct output 2 via traversing block FxStpRd : BOOL:=0; // EPOS-Wort-2 Bit 12 --> 1 = Fixed STOP reached FxStpTrRd : BOOL:=0; // EPOS-Wort-2 Bit 13 --> 1 = Fixed STOP clamping torque reached TrvFxStpAct : BOOL:=0; // EPOS-Wort-2 Bit 14 --> 1 = Traversing fixed STOP active CmdAct : BOOL:=0; // EPOS-Wort-2 Bit 15 --> 1 = Traversing command active TrkModeAct : BOOL:=0; // EPOS-Wort-2 Bit 00 --> 1 = Tracking mode active VeloLimAct : BOOL:=0; // EPOS-Wort-2 Bit 01 --> 1 = Velocity limit active SetPStat : BOOL:=0; // EPOS-Wort-2 Bit 02 --> 1 = Setpoint static PrnMrkOut : BOOL:=0; // EPOS-Wort-2 Bit 03 --> 1 = Printmark outside outer window FWD : BOOL:=0; // EPOS-Wort-2 Bit 04 --> 1 = Axis forwards BWD : BOOL:=0; // EPOS-Wort-2 Bit 05 --> 1 = Axis backwards SftSwMinAct : BOOL:=0; // EPOS-Wort-2 Bit 06 --> 1 = Software limit switch minus active SftSwPlsAct : BOOL:=0; // EPOS-Wort-2 Bit 07 --> 1 = Software limit switch plus active END_STRUCT;
         ZSW2 : Word := WORD#16#0000;   // ZSW2sxZSW2 : STRUCT Bit08 : BOOL:=0; // ZSW-Wort-2 Bit 08 --> Reserve GlbTrgReq : BOOL:=0; // ZSW-Wort-2 Bit 09 --> Global trigger request PulsEn : BOOL:=0; // ZSW-Wort-2 Bit 10 --> Pulses enabled MotSwOverAct : BOOL:=0; // ZSW-Wort-2 Bit 11 --> Motor switch over activ SlvZykBit0 : BOOL:=0; // ZSW-Wort-2 Bit 12 --> Slave - life bit 0 SlvZykBit1 : BOOL:=0; // ZSW-Wort-2 Bit 13 --> Slave - life bit 1 SlvZykBit2 : BOOL:=0; // ZSW-Wort-2 Bit 14 --> Slave - life bit 2 SlvZykBit3 : BOOL:=0; // ZSW-Wort-2 Bit 15 --> Slave - life bit 3 ActDDSBit0 : BOOL:=0; // ZSW-Wort-2 Bit 00 --> Active drive data set bit 0 ActDDSBit1 : BOOL:=0; // ZSW-Wort-2 Bit 01 --> Active drive data set bit 1 ActDDSBit2 : BOOL:=0; // ZSW-Wort-2 Bit 02 --> Active drive data set bit 2 ActDDSBit3 : BOOL:=0; // ZSW-Wort-2 Bit 03 --> Active drive data set bit 3 ActDDSBit4 : BOOL:=0; // ZSW-Wort-2 Bit 04 --> Active drive data set bit 4 CmdActRelBrk : BOOL:=0; // ZSW-Wort-2 Bit 05 --> Command "release holding break" active TrqContMode : BOOL:=0; // ZSW-Wort-2 Bit 06 --> Torque controlled mode ParkAxisAct : BOOL:=0; // ZSW-Wort-2 Bit 07 --> Parking axis activated END_STRUCT;
         NotUsed : Word := WORD#16#0000;   // Reserve
         Position : DWord := DWORD#16#0000_0000;   // Feedback of position
         Velocity : DWord := DWORD#16#0000_0000;   // Feedback of velocity
         ErrNr : Word := WORD#16#0000;   // Fault number
         WarnNr : Word := WORD#16#0000;   // Warning number
         Reserve : Word := WORD#16#0000;   // Reserve
      END_STRUCT;
      v1 : Real;
      v2 : Real;
   END_VAR
   VAR_TEMP
      piRetSFC : Int;   // Status for fault analysis
      piCount : Int;   // Freely available counter variable 3
      swSendBuf : Array[0..11] of Word;   // Send buffer
      swRecvBuf : Array[0..11] of Word;   // Receive buffer
      PositionDint : DInt;
      aaa : Real;
      bbb : Real;
      retval : Word;
   END_VAR
BEGIN

   //=============================================================================
   //SIEMENS AG
   //(c)Copyright 2019 All Rights Reserved
   //-----------------------------------------------------------------------------
   // Library: DriveLib
   // Tested with: -
   // Engineering: TIA Portal V15.1
   // Restrictions: -
   // Requirements: S7-1200 / S7-1500
   // Functionality: cyclic communication between a SINAMICS (Basic positioner)and a PLC
   //                If in HWConfig Std.TLG 111 is projected 12 PZD-words are exchanged
   //                in every bus cycle.
   //                The parametrisation of these words is described in the manual of the
   //                SINAMICS
   //=============================================================================
   #PositionDint := REAL_TO_DINT(#Position);
   // Betriebsart ermitteln
   IF #ModePos > #siModePosMax THEN

     #sbModePos := FALSE;
     #Error := True;
     #swStatus := 16#8202;
   ELSIF #ModePos < 1 THEN

     #sbModePos := FALSE;
     #Error := True;
     #swStatus := 16#8202;
   ELSE
     // Betriebsartenwechsel ist nur möglich, wenn die Achse nicht beschleunigt oder nicht verzögert 
     // und die Geschwindigkeit Null ist
     IF NOT #sbFWD AND NOT #sbBWD AND NOT #sbAccel AND NOT #sbDecel THEN

       #sbModePos := TRUE;
       #siModePos := #ModePos;

       // Fehler wieder zurücknehmen, wenn er mal ausgelöst wurde
       IF #swStatus = 16#8202 THEN
         #swStatus := 16#7002;
         #Error := False;
       END_IF;
     END_IF;
   END_IF;

   // Überprüfung der analogen Eingabewerte, ob sie innerhalb des möglichen Bereiches liegen
   // Geschwindigkeitsoverride (0% - 199%, 100% => W#16#4000)
   IF (#OverV < 0) OR (#OverV > 199) THEN
     #swStatus := 16#8203;
     #Error := True;
   ELSE
     // Geschwindigkeitsoverride in den Sendepuffer eintragen
     #sxSendBuf.OverrideV := INT_TO_WORD(REAL_TO_INT(16384.0 * (INT_TO_REAL(#OverV) / 100.0)));
   END_IF;

   // Beschleunigungsoverride (0% - 100%, 100% => W#16#4000)
   IF (#OverAcc < 0) OR (#OverAcc > 100) THEN
     #swStatus := 16#8203;
     #Error := True;
   ELSE
     // Beschleunigungsoverride in den Sendepuffer eintragen
     #sxSendBuf.OverrideA := INT_TO_WORD(REAL_TO_INT(16384.0 * (INT_TO_REAL(#OverAcc) / 100.0)));
   END_IF;

   // Verzögerungsoverride (0% - 100%, 100% => W#16#4000)
   IF (#OverDec < 0) OR (#OverDec > 100) THEN
     #swStatus := 16#8203;
     #Error := True;
   ELSE
     // Verzögerungsoverride in den Sendepuffer eintragen
     #sxSendBuf.OverrideD := INT_TO_WORD(REAL_TO_INT(16384.0 * (INT_TO_REAL(#OverDec) / 100.0)));
   END_IF;

   // Fehler wieder zurücknehmen, wenn er mal ausgelöst wurde
   IF NOT (#OverV < 0) AND NOT (#OverV > 199) AND NOT (#OverAcc < 0) AND NOT (#OverAcc > 100) AND
       NOT (#OverDec < 0) AND NOT (#OverDec > 100) THEN
       IF #swStatus = 16#8203 THEN
           #swStatus := 16#7002;
           #Error := False;
       END_IF;
   END_IF;

   // Positionssollwert
   // Positionssollwert in den Sendepuffer eintragen
   #sxSendBuf.Position := DINT_TO_DWORD(REAL_TO_DINT(#Position * #Factor));

   // Geschwindigkeitssollwert (Begrenzung / Überwachung
   // Geschwindigkeitssollwert in den Sendepuffer eintragen
   #sxSendBuf.Velocity := DINT_TO_DWORD(#Velocity);

   // Einschalten bzw. Ausschalten des Antriebes erkennen
   IF #EnableAxis AND NOT #sbOff1Edge AND NOT #sbBusy AND #sbModePos THEN
     #sbOff1 := True;
   END_IF;
   // Einschalten bzw. Ausschalten des Antriebes Flanke merken
   #sbOff1Edge := #EnableAxis AND NOT #sbBusy;

   // Einschaltflankenmerker wieder zurücksetzen
   IF NOT #EnableAxis THEN
     #sbOff1 := False;
   END_IF;

   // Fliegendes Referenzieren aktivieren erkennen
   IF #FlyRef AND NOT #sbRefTypEdge THEN
     #sbRefTyp := True;
   END_IF;
   // Fliegendes Referenzieren aktivieren Flanke merken
   #sbRefTypEdge := #FlyRef;

   // Fliegendes Referenzieren Flankenmerker wieder zurücksetzen
   IF NOT #FlyRef THEN
     #sbRefTyp := False;
     #siRefTypCyc := 0;
   END_IF;

   // Betriebsart aktivieren erkennen (RQ 3901129, RQ 4094299)
   IF #ExecuteMode AND NOT #sbExecuteEdge THEN
     #sbExecute := True;
     #siExecuteCyc := 0;
   ELSIF #ActMode <> #ModePos THEN
     #sbExecute := FALSE;
   ELSIF #siExecuteCyc > (2 * #siCycWait) THEN
     IF #ModePos <> 4 THEN
       #sbExecute := FALSE;
     ELSE
       IF #sxRecvBuf.ZSW1.%X11 OR NOT #ExecuteMode THEN
         #sbExecute := FALSE;
       END_IF;
     END_IF;
   ELSE
     ; // not used
   END_IF;

   IF #siExecuteCyc > 100 THEN
     #siExecuteCyc := 0;
   ELSE
     #siExecuteCyc := #siExecuteCyc + 1;
   END_IF;

   // Verfahrauftrag aktivieren Flanke merken
   #sbExecuteEdge := #ExecuteMode;

   // Betriebsart MDI / Sollwertdirektvorgabe Flanke merken
   (*IF #sxSendBuf.sxEPosSTW1.MdiStart AND NOT #sbMdiStartEdge THEN
             #sbMdiStart := True;
         END_IF;
         // Betriebsart MDI / Sollwertdirektvorgabe Flanke merken
         #sbMdiStartEdge := #sxSendBuf.sxEPosSTW1.MdiStart AND NOT #Busy;*)

   // Verfahrauftragflankenmerker wieder zurücksetzen
   (*IF NOT #sxSendBuf.sxEPosSTW1.MdiStart THEN
             #sbMdiStart := False;
             #siMdiStartCyc := 0;
         END_IF;*)

   IF #sxSendBuf.EPosSTW1.%X15 AND NOT #sbMdiStartEdge THEN
     #sbMdiStart := True;
   END_IF;
   // Betriebsart MDI / Sollwertdirektvorgabe Flanke merken
   #sbMdiStartEdge := #sxSendBuf.EPosSTW1.%X15 AND NOT #sbBusy;

   // Verfahrauftragflankenmerker wieder zurücksetzen
   IF NOT #sxSendBuf.EPosSTW1.%X15 THEN
     #sbMdiStart := False;
     #siMdiStartCyc := 0;
   END_IF;

   // Schreibdaten zusammenstellen
   // Steuerword STW1 für alle Betriebsart aufbereiten
   (*#sxSendBuf.sxSTW1.RejTrvTsk        := #RejTrvTsk;
         #sxSendBuf.sxSTW1.IntMStop         := #IntMStop;
         #sxSendBuf.sxSTW1.AckFault         := #AckFlt;*)

   #sxSendBuf.STW1.%X4 := #CancelTraversing;
   #sxSendBuf.STW1.%X5 := #IntermediateStop;
   #sxSendBuf.STW1.%X7 := #AckError;
   #sxSendBuf.STW1.%X1 := TRUE;
   #sxSendBuf.STW1.%X2 := TRUE;
   #sxSendBuf.STW1.%X3 := TRUE;
   #sxSendBuf.STW1.%X10 := TRUE;

   // Hauptbetriebsart "Positionieren / manueller Sollwertvorgabe (MDI)" 
   // Betriebsart "Positionieren Relativ positiv" oder "Positionieren Relativ negativ"
   IF (#siModePos = 1 AND #sbModePos) THEN

     // Antrieb einschalten
     //#sxSendBuf.sxSTW1.Off1 := #sbOff1;
     #sxSendBuf.STW1.%X0 := #sbOff1;

     // nicht verwendete Signale für den 1. Schritt und eventuell weitere Schritte
     (*#sxSendBuf.sxSTW1.Jog1          := False;
             #sxSendBuf.sxSTW1.Jog2          := False;
             #sxSendBuf.sxEPosSTW1.MdiTyp    := False;
             #sxSendBuf.sxEPosSTW1.MdiPos    := False;
             #sxSendBuf.sxEPosSTW1.MdiNeg    := False;
             #sxSendBuf.sxEPosSTW1.MdiSetup  := False;
             #sxSendBuf.sxEPosSTW2.SetRefPt  := False;
             #sxSendBuf.sxEPosSTW2.JogInc    := False;
             #sxSendBuf.sxEPosSTW2.RefStDi   := False;
             #sxSendBuf.sxSTW1.RefStart      := False;
             #sxSendBuf.sxEPosSTW2.RefTyp    := False;
             #sxSendBuf.sxEPosSTW1.MdiStart  := False;*)
     #sxSendBuf.STW1.%X8 := False;
     #sxSendBuf.STW1.%X9 := False;
     #sxSendBuf.EPosSTW1.%X8 := False;
     #sxSendBuf.EPosSTW1.%X9 := False;
     #sxSendBuf.EPosSTW1.%X10 := False;
     #sxSendBuf.EPosSTW1.%X14 := False;
     #sxSendBuf.EPosSTW2.%X1 := False;
     #sxSendBuf.EPosSTW2.%X5 := False;
     #sxSendBuf.EPosSTW2.%X9 := False;
     #sxSendBuf.STW1.%X11 := False;
     #sxSendBuf.EPosSTW2.%X8 := False;
     #sxSendBuf.EPosSTW1.%X15 := False;


     // Nach dem Einschalten des Antriebes, prüfen ob der Antrieb betriebsbereit, in Operation ohne Fehler und Warnung ist, 
     // dann die Betriebsart MDI / Sollwertvorgabe Start gesetzt werden
     IF #sbOff1 AND #sbReady AND #sbIOp AND NOT #sbFault THEN

       // Betriebsart MDI / Sollwertdirektvorgabe setzen
       //#sxSendBuf.sxEPosSTW1.MdiStart := True;
       #sxSendBuf.EPosSTW1.%X15 := True;

       // Positioniertyp auf relatives Positionieren stellen 
       //#sxSendBuf.sxEPosSTW1.MdiTyp := False;
       #sxSendBuf.EPosSTW1.%X8 := False;

       // die Richtungswahl für das Positionieren auf positive Richtung oder negative Richtung einstellen
       IF #Positive AND NOT #Negative THEN

         // positive Richtung
         //#sxSendBuf.sxEPosSTW1.MdiPos := True;
         #sxSendBuf.EPosSTW1.%X9 := True;

         // negative Richtung
         //#sxSendBuf.sxEPosSTW1.MdiNeg := False;
         #sxSendBuf.EPosSTW1.%X10 := False;

         // die Richtungswahl für das Positionieren auf negative Richtung einstellen                
       ELSIF NOT #Positive AND #Negative THEN

         // positive Richtung
         //#sxSendBuf.sxEPosSTW1.MdiPos := False;
         #sxSendBuf.EPosSTW1.%X9 := False;

         // negative Richtung
         //#sxSendBuf.sxEPosSTW1.MdiNeg := True;
         #sxSendBuf.EPosSTW1.%X10 := True;

         // die Richtungswahl für das Positionieren auf keine Richtung einstellen                
       ELSE

         // positive Richtung
         //#sxSendBuf.sxEPosSTW1.MdiPos := False;
         #sxSendBuf.EPosSTW1.%X9 := False;

         // negative Richtung
         //#sxSendBuf.sxEPosSTW1.MdiNeg := False;
         #sxSendBuf.EPosSTW1.%X10 := False;

       END_IF;

       // Nach dem Einschalten des Antriebes und dem Betriebsart MDI / Sollwertvorgabe starten, 
       // ein Paar Zyklen warten bevor die Flanke für die Sollwertübernahme MDI gesetzt werden kann
       IF #sbMdiStart AND (#siMdiStartCyc < #siCycWait) THEN
         #siMdiStartCyc := #siMdiStartCyc + 1;
       ELSE
         // Flanke Sollwertübernahme MDI
         //#sxSendBuf.sxSTW1.TrvStart := #Execute;
         #sxSendBuf.STW1.%X6 := #sbExecute;

       END_IF;

       // "Fliegendes Referentieren" aktivieren
       // "Fliegendes Referenzieren" erst nach Einschalten des Antriebes möglich
       IF #sbRefTyp THEN

         // Referenziertyp auf "Fliegendes Referenzieren" einstellen
         //#sxSendBuf.sxEPosSTW2.RefTyp := True;
         #sxSendBuf.EPosSTW2.%X8 := True;

         // Nach der Anwahl des Referenziertyps "Fliegendes Referenzieren", 
         // ein Zyklus später kann das Referenzieren gestartet
         IF (#siRefTypCyc = 0) THEN
           #siRefTypCyc := #siRefTypCyc + 1;
         ELSE
           // Referenzieren starten
           //#sxSendBuf.sxSTW1.RefStart := True;
           #sxSendBuf.STW1.%X11 := True;

         END_IF;
       END_IF;
     END_IF;

     // Betriebsart "Positionieren Absolut" oder "Positonieren Absolut positiv" oder "Positionieren Absolut negativ"
   ELSIF #siModePos = 2 AND #sbModePos THEN

     // Antrieb einschalten
     //#sxSendBuf.sxSTW1.Off1 := #sbOff1;
     #sxSendBuf.STW1.%X0 := #sbOff1;

     // nicht verwendete Signale für den 1. Schritt und eventuell weitere Schritte
     (*#sxSendBuf.sxSTW1.Jog1         := False;
             #sxSendBuf.sxSTW1.Jog2         := False;
             #sxSendBuf.sxEPosSTW1.MdiTyp   := False;
             #sxSendBuf.sxEPosSTW1.MdiPos   := False;
             #sxSendBuf.sxEPosSTW1.MdiNeg   := False;
             #sxSendBuf.sxEPosSTW1.MdiSetup := False;
             #sxSendBuf.sxEPosSTW2.SetRefPt := False;
             #sxSendBuf.sxEPosSTW2.JogInc   := False;
             #sxSendBuf.sxEPosSTW2.RefStDi  := False;
             #sxSendBuf.sxSTW1.RefStart     := False;
             #sxSendBuf.sxEPosSTW2.RefTyp   := False;
             #sxSendBuf.sxEPosSTW1.MdiStart := False;*)
     #sxSendBuf.STW1.%X8 := False;
     #sxSendBuf.STW1.%X9 := False;
     #sxSendBuf.EPosSTW1.%X8 := False;
     #sxSendBuf.EPosSTW1.%X9 := False;
     #sxSendBuf.EPosSTW1.%X10 := False;
     #sxSendBuf.EPosSTW1.%X14 := False;
     #sxSendBuf.EPosSTW2.%X1 := False;
     #sxSendBuf.EPosSTW2.%X5 := False;
     #sxSendBuf.EPosSTW2.%X9 := False;
     #sxSendBuf.STW1.%X11 := False;
     #sxSendBuf.EPosSTW2.%X8 := False;
     #sxSendBuf.EPosSTW1.%X15 := False;

     // Nach dem Einschalten des Antriebes, prüfen ob der Antrieb betriebsbereit, in Operation ohne Fehler und Warnung ist, 
     // dann die Betriebsart MDI / Sollwertvorgabe Start gesetzt werden
     IF #sbOff1 AND #sbReady AND #sbIOp AND NOT #sbFault THEN

       // Betriebsart MDI / Sollwertdirektvorgabe setzen
       //#sxSendBuf.sxEPosSTW1.MdiStart := True;
       #sxSendBuf.EPosSTW1.%X15 := True;

       // Positioniertyp auf absolutes Positionieren stellen 
       //#sxSendBuf.sxEPosSTW1.MdiTyp := True;
       #sxSendBuf.EPosSTW1.%X8 := True;

       // die Richtungswahl für das Positionieren auf positive Richtung oder negative Richtung einstellen
       IF #Positive AND NOT #Negative THEN

         // positive Richtung
         //#sxSendBuf.sxEPosSTW1.MdiPos := True;
         #sxSendBuf.EPosSTW1.%X9 := True;

         // negative Richtung
         //#sxSendBuf.sxEPosSTW1.MdiNeg := False;
         #sxSendBuf.EPosSTW1.%X10 := False;

         // die Richtungswahl für das Positionieren auf negative Richtung einstellen                
       ELSIF NOT #Positive AND #Negative THEN

         // positive Richtung
         //#sxSendBuf.sxEPosSTW1.MdiPos := False;
         #sxSendBuf.EPosSTW1.%X9 := False;

         // negative Richtung
         //#sxSendBuf.sxEPosSTW1.MdiNeg := True;
         #sxSendBuf.EPosSTW1.%X10 := True;

         // die Richtungswahl für das Positionieren auf keine Richtung einstellen                
       ELSE

         // positive Richtung
         //#sxSendBuf.sxEPosSTW1.MdiPos := False;
         #sxSendBuf.EPosSTW1.%X9 := False;

         // negative Richtung
         //#sxSendBuf.sxEPosSTW1.MdiNeg := False;
         #sxSendBuf.EPosSTW1.%X10 := False;

       END_IF;

       // Nach dem Einschalten des Antriebes und dem Betriebsart MDI / Sollwertvorgabe starten, 
       // ein Paar Zyklen warten bevor die Flanke für die Sollwertübernahme MDI gesetzt werden kann
       IF #sbMdiStart AND (#siMdiStartCyc < #siCycWait) THEN
         #siMdiStartCyc := #siMdiStartCyc + 1;
       ELSE
         // Flanke Sollwertübernahme MDI
         //#sxSendBuf.sxSTW1.TrvStart := #Execute;
         #sxSendBuf.STW1.%X6 := #sbExecute;

       END_IF;

       // "Fliegendes Referentieren" aktivieren
       // "Fliegendes Referenzieren" erst nach Einschalten des Antriebes möglich
       IF #sbRefTyp THEN

         // Referenziertyp auf "Fliegendes Referenzieren" einstellen
         //#sxSendBuf.sxEPosSTW2.RefTyp := True;
         #sxSendBuf.EPosSTW2.%X8 := True;

         // Nach der Anwahl des Referenziertyps "Fliegendes Referenzieren", 
         // ein Zyklus später kann das Referenzieren gestartet
         IF (#siRefTypCyc = 0) THEN
           #siRefTypCyc := #siRefTypCyc + 1;
         ELSE
           // Referenzieren starten
           //#sxSendBuf.sxSTW1.RefStart := True;
           #sxSendBuf.STW1.%X11 := True;

         END_IF;
       END_IF;
     END_IF;

     // Betriebsart "Positionieren als Einrichten positiv" oder "Positionieren als Einrichten negativ"
   ELSIF #siModePos = 3 AND #sbModePos THEN

     // Antrieb einschalten
     //#sxSendBuf.sxSTW1.Off1 := #sbOff1;
     #sxSendBuf.STW1.%X0 := #sbOff1;

     // nicht verwendete Signale für den 1. Schritt und eventuell weitere Schritte
     (*#sxSendBuf.sxSTW1.Jog1           := False;
             #sxSendBuf.sxSTW1.Jog2           := False;
             #sxSendBuf.sxEPosSTW1.MdiTyp     := False;
             #sxSendBuf.sxEPosSTW1.MdiPos     := False;
             #sxSendBuf.sxEPosSTW1.MdiNeg     := False;
             #sxSendBuf.sxEPosSTW1.MdiSetup   := False;
             #sxSendBuf.sxEPosSTW2.SetRefPt   := False;
             #sxSendBuf.sxEPosSTW2.JogInc     := False;
             #sxSendBuf.sxEPosSTW2.RefStDi    := False;
             #sxSendBuf.sxSTW1.RefStart       := False;
             #sxSendBuf.sxEPosSTW2.RefTyp     := False;
             #sxSendBuf.sxEPosSTW1.MdiStart   := False;*)
     #sxSendBuf.STW1.%X8 := False;
     #sxSendBuf.STW1.%X9 := False;
     #sxSendBuf.EPosSTW1.%X8 := False;
     #sxSendBuf.EPosSTW1.%X9 := False;
     #sxSendBuf.EPosSTW1.%X10 := False;
     #sxSendBuf.EPosSTW1.%X14 := False;
     #sxSendBuf.EPosSTW2.%X1 := False;
     #sxSendBuf.EPosSTW2.%X5 := False;
     #sxSendBuf.EPosSTW2.%X9 := False;
     #sxSendBuf.STW1.%X11 := False;
     #sxSendBuf.EPosSTW2.%X8 := False;
     #sxSendBuf.EPosSTW1.%X15 := False;

     // Nach dem Einschalten des Antriebes, prüfen ob der Antrieb betriebsbereit, in Operation ohne Fehler und Warnung ist, 
     // dann die Betriebsart MDI / Sollwertvorgabe Start gesetzt werden
     IF #sbOff1 AND #sbReady AND #sbIOp AND NOT #sbFault THEN

       // Betriebsart MDI / Sollwertdirektvorgabe setzen
       //#sxSendBuf.sxEPosSTW1.MdiStart := True;
       #sxSendBuf.EPosSTW1.%X15 := True;

       // Positioniertyp auf absolutes Positionieren stellen 
       //#sxSendBuf.sxEPosSTW1.MdiTyp := True;
       #sxSendBuf.EPosSTW1.%X8 := True;

       // die Anwahl für MDI Modus auf Einrichten einstellen
       //#sxSendBuf.sxEPosSTW1.MdiSetup := True;
       #sxSendBuf.EPosSTW1.%X14 := True;

       // die Richtungswahl für das Positionieren auf positive Richtung oder negative Richtung einstellen
       IF #Positive AND NOT #Negative THEN

         // positive Richtung
         //#sxSendBuf.sxEPosSTW1.MdiPos := True;
         #sxSendBuf.EPosSTW1.%X9 := True;

         // negative Richtung
         //#sxSendBuf.sxEPosSTW1.MdiNeg := False;
         #sxSendBuf.EPosSTW1.%X10 := False;

         // die Richtungswahl für das Positionieren auf negative Richtung einstellen                
       ELSIF NOT #Positive AND #Negative THEN

         // positive Richtung
         //#sxSendBuf.sxEPosSTW1.MdiPos := False;
         #sxSendBuf.EPosSTW1.%X9 := False;

         // negative Richtung
         //#sxSendBuf.sxEPosSTW1.MdiNeg := True;
         #sxSendBuf.EPosSTW1.%X10 := True;

         // die Richtungswahl für das Positionieren auf keine Richtung einstellen                
       ELSE

         // positive Richtung
         //#sxSendBuf.sxEPosSTW1.MdiPos := False;
         #sxSendBuf.EPosSTW1.%X9 := False;

         // negative Richtung
         //#sxSendBuf.sxEPosSTW1.MdiNeg := False;
         #sxSendBuf.EPosSTW1.%X10 := False;

       END_IF;

       // Nach dem Einschalten des Antriebes und dem Betriebsart MDI / Sollwertvorgabe starten, 
       // ein Paar Zyklen warten bevor die Flanke für die Sollwertübernahme MDI gesetzt werden kann
       IF #sbMdiStart AND (#siMdiStartCyc < #siCycWait) THEN
         #siMdiStartCyc := #siMdiStartCyc + 1;
       ELSE
         // Flanke Sollwertübernahme MDI
         //#sxSendBuf.sxSTW1.TrvStart := #Execute;
         #sxSendBuf.STW1.%X6 := #sbExecute;

       END_IF;

       // "Fliegendes Referentieren" aktivieren
       // "Fliegendes Referenzieren" erst nach Einschalten des Antriebes möglich
       IF #sbRefTyp THEN

         // Referenziertyp auf "Fliegendes Referenzieren" einstellen
         //#sxSendBuf.sxEPosSTW2.RefTyp := True;
         #sxSendBuf.EPosSTW2.%X8 := True;

         // Nach der Anwahl des Referenziertyps "Fliegendes Referenzieren", 
         // ein Zyklus später kann das Referenzieren gestartet
         IF (#siRefTypCyc = 0) THEN
           #siRefTypCyc := #siRefTypCyc + 1;
         ELSE
           // Referenzieren starten
           //#sxSendBuf.sxSTW1.RefStart := True;
           #sxSendBuf.STW1.%X11 := True;

         END_IF;
       END_IF;
     END_IF;

     // Hauptbetriebsart "Referenzieren" (Reference)
     // Betriebsart "Referenzieren - Referenzpunktfahrt positiv" oder "Referenzieren - Referenzpunktfahrt negativ"
   ELSIF #siModePos = 4 AND #sbModePos THEN

     // Antrieb einschalten
     //#sxSendBuf.sxSTW1.Off1 := #sbOff1;
     #sxSendBuf.STW1.%X0 := #sbOff1;

     // nicht verwendete Signale für den 1. Schritt und eventuell weitere Schritte
     (*#sxSendBuf.sxSTW1.Jog1         := False;
             #sxSendBuf.sxSTW1.Jog2         := False;
             #sxSendBuf.sxEPosSTW1.MdiStart := False;
             #sxSendBuf.sxEPosSTW2.SetRefPt := False;
             #sxSendBuf.sxEPosSTW2.JogInc   := False;
             #sxSendBuf.sxEPosSTW2.RefTyp   := False;
             #sxSendBuf.sxSTW1.RefStart     := False;
             #sxSendBuf.sxEPosSTW2.RefStDi  := False;*)
     #sxSendBuf.STW1.%X8 := False;
     #sxSendBuf.STW1.%X9 := False;
     #sxSendBuf.EPosSTW1.%X15 := False;
     #sxSendBuf.EPosSTW2.%X1 := False;
     #sxSendBuf.EPosSTW2.%X5 := False;
     #sxSendBuf.EPosSTW2.%X8 := False;
     #sxSendBuf.STW1.%X11 := False;
     #sxSendBuf.EPosSTW2.%X9 := False;

     // Nach dem Einschalten des Antriebes, prüfen ob der Antrieb betriebsbereit, in Operation ohne Fehler und Warnung ist, 
     // dann die Betriebsart MDI / Sollwertvorgabe Start gesetzt werden
     IF #sbOff1 AND #sbReady AND #sbIOp AND NOT #sbFault THEN

       // Referenzieren starten
       //#sxSendBuf.sxSTW1.RefStart := #Execute;
       #sxSendBuf.STW1.%X11 := #sbExecute;

       // die Richtungswahl für das Referenzpunktfahrt positiv einstellen
       IF #Positive AND NOT #Negative THEN

         // positive Referenzpunktfahrt
         //#sxSendBuf.sxEPosSTW2.RefStDi := False;
         #sxSendBuf.EPosSTW2.%X9 := False;

         // die Richtungswahl für das Referenzpunktfahrt negativ einstellen                
       ELSIF NOT #Positive AND #Negative THEN

         // negative Referenzpunktfahrt
         //#sxSendBuf.sxEPosSTW2.RefStDi := True;
         #sxSendBuf.EPosSTW2.%X9 := True;

       END_IF;
     END_IF;

     // Betriebsart "Referenzieren - Referenzpunkt setzen"
   ELSIF #siModePos = 5 AND #sbModePos THEN

     // Antrieb einschalten
     //#sxSendBuf.sxSTW1.Off1 := #sbOff1;
     #sxSendBuf.STW1.%X0 := #sbOff1;

     // nicht verwendete Signale für den 1. Schritt und eventuell weitere Schritte
     (*#sxSendBuf.sxSTW1.Jog1          := False;
             #sxSendBuf.sxSTW1.Jog2          := False;
             #sxSendBuf.sxSTW1.RefStart      := False;
             #sxSendBuf.sxEPosSTW1.MdiStart  := False;
             #sxSendBuf.sxEPosSTW2.JogInc    := False;
             #sxSendBuf.sxEPosSTW2.RefTyp    := False;
             #sxSendBuf.sxEPosSTW2.RefStDi   := False;
             #sxSendBuf.sxEPosSTW2.SetRefPt  := False;*)
     #sxSendBuf.STW1.%X8 := False;
     #sxSendBuf.STW1.%X9 := False;
     #sxSendBuf.STW1.%X11 := False;
     #sxSendBuf.EPosSTW1.%X15 := False;
     #sxSendBuf.EPosSTW2.%X5 := False;
     #sxSendBuf.EPosSTW2.%X8 := False;
     #sxSendBuf.EPosSTW2.%X9 := False;
     #sxSendBuf.EPosSTW2.%X1 := False;

     // Nach dem Einschalten des Antriebes, prüfen ob der Antrieb betriebsbereit, in Operation ohne Fehler und Warnung ist, 
     // dann die Betriebsart MDI / Sollwertvorgabe Start gesetzt werden
     IF NOT #sbFault THEN

       // Referenzpunktfahrt negativ
       //#sxSendBuf.sxEPosSTW2.SetRefPt := #Execute;
       #sxSendBuf.EPosSTW2.%X1 := #sbExecute;

     END_IF;

     // Hauptbetriebsart "Verfahrsätze" (Traversing Blocks)
   ELSIF #siModePos = 6 AND #sbModePos THEN

     // Antrieb einschalten
     //#sxSendBuf.sxSTW1.Off1 := #sbOff1;
     #sxSendBuf.STW1.%X0 := #sbOff1;

     // nicht verwendete Signale für den 1. Schritt und eventuell weitere Schritte
     (*#sxSendBuf.sxSTW1.Jog1          := False;
             #sxSendBuf.sxSTW1.Jog2          := False;
             #sxSendBuf.sxEPosSTW1.MdiTyp    := False;
             #sxSendBuf.sxEPosSTW1.MdiPos    := False;
             #sxSendBuf.sxEPosSTW1.MdiNeg    := False;
             #sxSendBuf.sxEPosSTW1.MdiSetup  := False;
             #sxSendBuf.sxEPosSTW2.SetRefPt  := False;
             #sxSendBuf.sxEPosSTW2.JogInc    := False;
             #sxSendBuf.sxEPosSTW2.RefStDi   := False;
             #sxSendBuf.sxEPosSTW2.RefTyp    := False;
             #sxSendBuf.sxSTW1.RefStart      := False;
             #sxSendBuf.sxEPosSTW1.TrvBit0   := False;
             #sxSendBuf.sxEPosSTW1.TrvBit1   := False;
             #sxSendBuf.sxEPosSTW1.TrvBit2   := False;
             #sxSendBuf.sxEPosSTW1.TrvBit3   := False;
             #sxSendBuf.sxEPosSTW1.TrvBit4   := False;
             #sxSendBuf.sxEPosSTW1.TrvBit5   := False;
             #sxSendBuf.sxEPosSTW1.MdiStart  := False;*)
     #sxSendBuf.STW1.%X8 := False;
     #sxSendBuf.STW1.%X9 := False;
     #sxSendBuf.EPosSTW1.%X8 := False;
     #sxSendBuf.EPosSTW1.%X9 := False;
     #sxSendBuf.EPosSTW1.%X10 := False;
     #sxSendBuf.EPosSTW1.%X14 := False;
     #sxSendBuf.EPosSTW2.%X1 := False;
     #sxSendBuf.EPosSTW2.%X5 := False;
     #sxSendBuf.EPosSTW2.%X9 := False;
     #sxSendBuf.EPosSTW2.%X8 := False;
     #sxSendBuf.STW1.%X11 := False;
     #sxSendBuf.EPosSTW1.%X0 := False;
     #sxSendBuf.EPosSTW1.%X1 := False;
     #sxSendBuf.EPosSTW1.%X2 := False;
     #sxSendBuf.EPosSTW1.%X3 := False;
     #sxSendBuf.EPosSTW1.%X4 := False;
     #sxSendBuf.EPosSTW1.%X5 := False;
     #sxSendBuf.EPosSTW1.%X15 := False;

     // Bei der Auswahl der Verfahrsätze entspricht die Position der Verfahrensatznummer 
     // Verfahrsatznummer aus der Position ermitteln und in die einzelnen Bit's aufteilen
     // Es sind die Verfahrsatznummern 0 - 63 möglich
     IF (DINT_TO_INT(#PositionDint) < 0) OR (DINT_TO_INT(#PositionDint) > 63) THEN
       // Fehler, ungültiger Verfahrsatznummer
       #swStatus := 16#8204;
       #Error := True;
     ELSE
       // Fehler wieder zurücknehmen, wenn er mal ausgelöst wurde
       IF #swStatus = 16#8204 THEN
         #swStatus := 16#7002;
         #Error := False;
       END_IF;

       // Verfahrsatznummer Bit 0 ermitteln
       IF (DINT_TO_WORD(#PositionDint) AND W#16#01) = W#16#01 THEN
         //#sxSendBuf.sxEPosSTW1.TrvBit0 := True;
         #sxSendBuf.EPosSTW1.%X0 := True;
       END_IF;

       // Verfahrsatznummer Bit 1 ermitteln
       IF (DINT_TO_WORD(#PositionDint) AND W#16#02) = W#16#02 THEN
         //#sxSendBuf.sxEPosSTW1.TrvBit1 := True;
         #sxSendBuf.EPosSTW1.%X1 := True;
       END_IF;

       // Verfahrsatznummer Bit 2 ermitteln
       IF (DINT_TO_WORD(#PositionDint) AND W#16#04) = W#16#04 THEN
         //#sxSendBuf.sxEPosSTW1.TrvBit2 := True;
         #sxSendBuf.EPosSTW1.%X2 := True;
       END_IF;

       // Verfahrsatznummer Bit 3 ermitteln
       IF (DINT_TO_WORD(#PositionDint) AND W#16#08) = W#16#08 THEN
         //#sxSendBuf.sxEPosSTW1.TrvBit3 := True;
         #sxSendBuf.EPosSTW1.%X3 := True;
       END_IF;

       // Verfahrsatznummer Bit 4 ermitteln
       IF (DINT_TO_WORD(#PositionDint) AND W#16#10) = W#16#10 THEN
         //#sxSendBuf.sxEPosSTW1.TrvBit4 := True;
         #sxSendBuf.EPosSTW1.%X4 := True;
       END_IF;

       // Verfahrsatznummer Bit 5 ermitteln
       IF (DINT_TO_WORD(#PositionDint) AND W#16#20) = W#16#20 THEN
         //#sxSendBuf.sxEPosSTW1.TrvBit5 := True;
         #sxSendBuf.EPosSTW1.%X5 := True;
       END_IF;

       // Nach dem Einschalten des Antriebes, prüfen ob der Antrieb betriebsbereit, in Operation ohne Fehler und Warnung ist, 
       // dann die Betriebsart MDI / Sollwertvorgabe Start gesetzt werden
       IF #sbOff1 AND #sbReady AND #sbIOp AND NOT #sbFault THEN

         #sxSendBuf.STW1.%X6 := #sbExecute;

         // "Fliegendes Referentieren" aktivieren
         // "Fliegendes Referenzieren" erst nach Einschalten des Antriebes möglich
         IF #sbRefTyp THEN

           // Referenziertyp auf "Fliegendes Referenzieren" einstellen
           //#sxSendBuf.sxEPosSTW2.RefTyp := True;
           #sxSendBuf.EPosSTW2.%X8 := True;

           // Nach der Anwahl des Referenziertyps "Fliegendes Referenzieren", 
           // ein Zyklus später kann das Referenzieren gestartet
           IF (#siRefTypCyc = 0) THEN
             #siRefTypCyc := #siRefTypCyc + 1;
           ELSE
             // Referenzieren starten
             //#sxSendBuf.sxSTW1.RefStart := True;
             #sxSendBuf.STW1.%X11 := True;
           END_IF;
         END_IF;
       END_IF;
     END_IF;

     // Hauptbetriebsart "Tippen" (Jogging)
     // Betriebsart "Tippen positiv" oder "Tippen negativ" angewählt 
   ELSIF #siModePos = 7 AND #sbModePos THEN

     // Antrieb einschalten
     //#sxSendBuf.sxSTW1.Off1 := #sbOff1;
     #sxSendBuf.STW1.%X0 := #sbOff1;

     // nicht verwendete Signale für den 1. Schritt und eventuell weitere Schritte
     (*#sxSendBuf.sxEPosSTW1.MdiStart := False;
             #sxSendBuf.sxEPosSTW2.JogInc   := False;
             #sxSendBuf.sxSTW1.Jog1         := False;
             #sxSendBuf.sxSTW1.Jog2         := False;
             #sxSendBuf.sxEPosSTW2.RefTyp   := False;
             #sxSendBuf.sxSTW1.RefStart     := False;
             #sxSendBuf.sxEPosSTW2.SetRefPt  := False;*)

     #sxSendBuf.EPosSTW1.%X15 := False;
     #sxSendBuf.EPosSTW2.%X5 := False;
     #sxSendBuf.STW1.%X8 := False;
     #sxSendBuf.STW1.%X9 := False;
     #sxSendBuf.EPosSTW2.%X8 := False;
     #sxSendBuf.STW1.%X11 := False;
     #sxSendBuf.EPosSTW2.%X1 := False;

     // Nach dem Einschalten des Antriebes, prüfen ob der Antrieb betriebsbereit, in Operation ohne Fehler und Warnung ist, 
     // dann kann Tippen positiv oder negativ gesetzt werden
     IF #sbOff1 AND #sbReady AND #sbIOp AND NOT #sbFault THEN

       // Tippen positiv
       IF #Jog1 AND NOT #Jog2 THEN
         //#sxSendBuf.sxSTW1.Jog1 := True;
         #sxSendBuf.STW1.%X8 := True;
       END_IF;

       // Tippen negativ
       IF #Jog2 AND NOT #Jog1 THEN
         //#sxSendBuf.sxSTW1.Jog2 := True;
         #sxSendBuf.STW1.%X9 := True;
       END_IF;

       // "Fliegendes Referentieren" aktivieren
       // "Fliegendes Referenzieren" erst nach Einschalten des Antriebes möglich
       IF #sbRefTyp THEN

         // Referenziertyp auf "Fliegendes Referenzieren" einstellen
         //#sxSendBuf.sxEPosSTW2.RefTyp := #FlyRef;
         #sxSendBuf.EPosSTW2.%X8 := #FlyRef;

         // Nach der Anwahl des Referenziertyps "Fliegendes Referenzieren", 
         // ein Zyklus später kann das Referenzieren gestartet
         IF (#siRefTypCyc = 0) THEN
           #siRefTypCyc := #siRefTypCyc + 1;
         ELSE
           // Referenzieren starten
           //#sxSendBuf.sxSTW1.RefStart := True;
           #sxSendBuf.STW1.%X11 := True;
         END_IF;
       END_IF;
     END_IF;

     // Betriebsart "Tippen positiv / Tippen negativ inkrementell" 
   ELSIF #siModePos = 8 AND #sbModePos THEN

     // Antrieb einschalten
     //#sxSendBuf.sxSTW1.OFF1 := #sbOff1;
     #sxSendBuf.STW1.%X0 := #sbOff1;

     // nicht verwendete Signale für den 1. Schritt und eventuell weitere Schritte
     (*#sxSendBuf.sxEPosSTW1.MdiStart := False;
             #sxSendBuf.sxEPosSTW2.JogInc   := False;
             #sxSendBuf.sxSTW1.Jog1         := False;
             #sxSendBuf.sxSTW1.Jog2         := False;
             #sxSendBuf.sxSTW1.RefStart     := False;
             #sxSendBuf.sxEPosSTW2.RefTyp   := False;
             #sxSendBuf.sxEPosSTW2.SetRefPt  := False;*)

     #sxSendBuf.EPosSTW1.%X15 := False;
     #sxSendBuf.EPosSTW2.%X5 := False;
     #sxSendBuf.STW1.%X8 := False;
     #sxSendBuf.STW1.%X9 := False;
     #sxSendBuf.STW1.%X11 := False;
     #sxSendBuf.EPosSTW2.%X8 := False;
     #sxSendBuf.EPosSTW2.%X1 := False;

     // Nach dem Einschalten des Antriebes, ein Paar Zyklen warten bevor Tippen negativ gesetzt werden kann
     // Nach dem Einschalten des Antriebes, prüfen ob der Antrieb betriebsbereit, in Operation ohne Fehler und Warnung ist, 
     // dann kann Tippen positiv oder negativ gesetzt werden
     IF #sbOff1 AND #sbReady AND #sbIOp AND NOT #sbFault THEN

       // Tippen inkrementell einstellen
       //#sxSendBuf.sxEPosSTW2.JogInc := True;
       #sxSendBuf.EPosSTW2.%X5 := True;

       #sbJogInc := True;

       // Nach dem Einstellen des Antriebes, ein Paar Zyklen warten bevor Tippen negativ oder Tippen positiv gesetz werden kann
       IF #sbJogInc AND (#siJogIncCyc = 0) THEN
         #siJogIncCyc := #siJogIncCyc + 1;
       ELSE

         // Tippen positiv oder negativ inkrementell zulassen
         IF #Jog1 XOR #Jog2 THEN

           //#sxSendBuf.sxSTW1.Jog1 := #Jog1;
           //#sxSendBuf.sxSTW1.Jog2 := #Jog2;
           #sxSendBuf.STW1.%X8 := #Jog1;
           #sxSendBuf.STW1.%X9 := #Jog2;
         END_IF;
       END_IF;

       // "Fliegendes Referentieren" aktivieren
       // "Fliegendes Referenzieren" erst nach Einschalten des Antriebes möglich
       IF #sbRefTyp THEN

         // Referenziertyp auf "Fliegendes Referenzieren" einstellen
         //#sxSendBuf.sxEPosSTW2.RefTyp := True;
         #sxSendBuf.EPosSTW2.%X8 := True;

